   // GBK_TO_UNICODE[4429] := 16#5C32;
   // GBK_TO_UNICODE[4430] := 16#8CBD;
   // GBK_TO_UNICODE[4431] := 16#5C33;
   // GBK_TO_UNICODE[4432] := 16#8CBE;
   // GBK_TO_UNICODE[4433] := 16#5C35;
   // GBK_TO_UNICODE[4434] := 16#8CBF;
   // GBK_TO_UNICODE[4435] := 16#5C36;
   // GBK_TO_UNICODE[4436] := 16#8CC0;
   // GBK_TO_UNICODE[4437] := 16#5C37;
   // GBK_TO_UNICODE[4438] := 16#8CC1;
   // GBK_TO_UNICODE[4439] := 16#5C43;
   // GBK_TO_UNICODE[4440] := 16#8CC2;
   // GBK_TO_UNICODE[4441] := 16#5C44;
   // GBK_TO_UNICODE[4442] := 16#8CC3;
   // GBK_TO_UNICODE[4443] := 16#5C46;
   // GBK_TO_UNICODE[4444] := 16#8CC4;
   // GBK_TO_UNICODE[4445] := 16#5C47;
   // GBK_TO_UNICODE[4446] := 16#8CC5;
   // GBK_TO_UNICODE[4447] := 16#5C4C;
   // GBK_TO_UNICODE[4448] := 16#8CC6;
   // GBK_TO_UNICODE[4449] := 16#5C4D;
   // GBK_TO_UNICODE[4450] := 16#8CC7;
   // GBK_TO_UNICODE[4451] := 16#5C52;
   // GBK_TO_UNICODE[4452] := 16#8CC8;
   // GBK_TO_UNICODE[4453] := 16#5C53;
   // GBK_TO_UNICODE[4454] := 16#8CC9;
   // GBK_TO_UNICODE[4455] := 16#5C54;
   // GBK_TO_UNICODE[4456] := 16#8CCA;
   // GBK_TO_UNICODE[4457] := 16#5C56;
   // GBK_TO_UNICODE[4458] := 16#8CCB;
   // GBK_TO_UNICODE[4459] := 16#5C57;
   // GBK_TO_UNICODE[4460] := 16#8CCC;
   // GBK_TO_UNICODE[4461] := 16#5C58;
   // GBK_TO_UNICODE[4462] := 16#8CCD;
   // GBK_TO_UNICODE[4463] := 16#5C5A;
   // GBK_TO_UNICODE[4464] := 16#8CCE;
   // GBK_TO_UNICODE[4465] := 16#5C5B;
   // GBK_TO_UNICODE[4466] := 16#8CCF;
   // GBK_TO_UNICODE[4467] := 16#5C5C;
   // GBK_TO_UNICODE[4468] := 16#8CD0;
   // GBK_TO_UNICODE[4469] := 16#5C5D;
   // GBK_TO_UNICODE[4470] := 16#8CD1;
   // GBK_TO_UNICODE[4471] := 16#5C5F;
   // GBK_TO_UNICODE[4472] := 16#8CD2;
   // GBK_TO_UNICODE[4473] := 16#5C62;
   // GBK_TO_UNICODE[4474] := 16#8CD3;
   // GBK_TO_UNICODE[4475] := 16#5C64;
   // GBK_TO_UNICODE[4476] := 16#8CD4;
   // GBK_TO_UNICODE[4477] := 16#5C67;
   // GBK_TO_UNICODE[4478] := 16#8CD5;
   // GBK_TO_UNICODE[4479] := 16#5C68;
   // GBK_TO_UNICODE[4480] := 16#8CD6;
   // GBK_TO_UNICODE[4481] := 16#5C69;
   // GBK_TO_UNICODE[4482] := 16#8CD7;
   // GBK_TO_UNICODE[4483] := 16#5C6A;
   // GBK_TO_UNICODE[4484] := 16#8CD8;
   // GBK_TO_UNICODE[4485] := 16#5C6B;
   // GBK_TO_UNICODE[4486] := 16#8CD9;
   // GBK_TO_UNICODE[4487] := 16#5C6C;
   // GBK_TO_UNICODE[4488] := 16#8CDA;
   // GBK_TO_UNICODE[4489] := 16#5C6D;
   // GBK_TO_UNICODE[4490] := 16#8CDB;
   // GBK_TO_UNICODE[4491] := 16#5C70;
   // GBK_TO_UNICODE[4492] := 16#8CDC;
   // GBK_TO_UNICODE[4493] := 16#5C72;
   // GBK_TO_UNICODE[4494] := 16#8CDD;
   // GBK_TO_UNICODE[4495] := 16#5C73;
   // GBK_TO_UNICODE[4496] := 16#8CDE;
   // GBK_TO_UNICODE[4497] := 16#5C74;
   // GBK_TO_UNICODE[4498] := 16#8CDF;
   // GBK_TO_UNICODE[4499] := 16#5C75;
   // GBK_TO_UNICODE[4500] := 16#8CE0;
   // GBK_TO_UNICODE[4501] := 16#5C76;
   // GBK_TO_UNICODE[4502] := 16#8CE1;
   // GBK_TO_UNICODE[4503] := 16#5C77;
   // GBK_TO_UNICODE[4504] := 16#8CE2;
   // GBK_TO_UNICODE[4505] := 16#5C78;
   // GBK_TO_UNICODE[4506] := 16#8CE3;
   // GBK_TO_UNICODE[4507] := 16#5C7B;
   // GBK_TO_UNICODE[4508] := 16#8CE4;
   // GBK_TO_UNICODE[4509] := 16#5C7C;
   // GBK_TO_UNICODE[4510] := 16#8CE5;
   // GBK_TO_UNICODE[4511] := 16#5C7D;
   // GBK_TO_UNICODE[4512] := 16#8CE6;
   // GBK_TO_UNICODE[4513] := 16#5C7E;
   // GBK_TO_UNICODE[4514] := 16#8CE7;
   // GBK_TO_UNICODE[4515] := 16#5C80;
   // GBK_TO_UNICODE[4516] := 16#8CE8;
   // GBK_TO_UNICODE[4517] := 16#5C83;
   // GBK_TO_UNICODE[4518] := 16#8CE9;
   // GBK_TO_UNICODE[4519] := 16#5C84;
   // GBK_TO_UNICODE[4520] := 16#8CEA;
   // GBK_TO_UNICODE[4521] := 16#5C85;
   // GBK_TO_UNICODE[4522] := 16#8CEB;
   // GBK_TO_UNICODE[4523] := 16#5C86;
   // GBK_TO_UNICODE[4524] := 16#8CEC;
   // GBK_TO_UNICODE[4525] := 16#5C87;
   // GBK_TO_UNICODE[4526] := 16#8CED;
   // GBK_TO_UNICODE[4527] := 16#5C89;
   // GBK_TO_UNICODE[4528] := 16#8CEE;
   // GBK_TO_UNICODE[4529] := 16#5C8A;
   // GBK_TO_UNICODE[4530] := 16#8CEF;
   // GBK_TO_UNICODE[4531] := 16#5C8B;
   // GBK_TO_UNICODE[4532] := 16#8CF0;
   // GBK_TO_UNICODE[4533] := 16#5C8E;
   // GBK_TO_UNICODE[4534] := 16#8CF1;
   // GBK_TO_UNICODE[4535] := 16#5C8F;
   // GBK_TO_UNICODE[4536] := 16#8CF2;
   // GBK_TO_UNICODE[4537] := 16#5C92;
   // GBK_TO_UNICODE[4538] := 16#8CF3;
   // GBK_TO_UNICODE[4539] := 16#5C93;
   // GBK_TO_UNICODE[4540] := 16#8CF4;
   // GBK_TO_UNICODE[4541] := 16#5C95;
   // GBK_TO_UNICODE[4542] := 16#8CF5;
   // GBK_TO_UNICODE[4543] := 16#5C9D;
   // GBK_TO_UNICODE[4544] := 16#8CF6;
   // GBK_TO_UNICODE[4545] := 16#5C9E;
   // GBK_TO_UNICODE[4546] := 16#8CF7;
   // GBK_TO_UNICODE[4547] := 16#5C9F;
   // GBK_TO_UNICODE[4548] := 16#8CF8;
   // GBK_TO_UNICODE[4549] := 16#5CA0;
   // GBK_TO_UNICODE[4550] := 16#8CF9;
   // GBK_TO_UNICODE[4551] := 16#5CA1;
   // GBK_TO_UNICODE[4552] := 16#8CFA;
   // GBK_TO_UNICODE[4553] := 16#5CA4;
   // GBK_TO_UNICODE[4554] := 16#8CFB;
   // GBK_TO_UNICODE[4555] := 16#5CA5;
   // GBK_TO_UNICODE[4556] := 16#8CFC;
   // GBK_TO_UNICODE[4557] := 16#5CA6;
   // GBK_TO_UNICODE[4558] := 16#8CFD;
   // GBK_TO_UNICODE[4559] := 16#5CA7;
   // GBK_TO_UNICODE[4560] := 16#8CFE;
   // GBK_TO_UNICODE[4561] := 16#5CA8;
   // GBK_TO_UNICODE[4562] := 16#8D40;
   // GBK_TO_UNICODE[4563] := 16#5CAA;
   // GBK_TO_UNICODE[4564] := 16#8D41;
   // GBK_TO_UNICODE[4565] := 16#5CAE;
   // GBK_TO_UNICODE[4566] := 16#8D42;
   // GBK_TO_UNICODE[4567] := 16#5CAF;
   // GBK_TO_UNICODE[4568] := 16#8D43;
   // GBK_TO_UNICODE[4569] := 16#5CB0;
   // GBK_TO_UNICODE[4570] := 16#8D44;
   // GBK_TO_UNICODE[4571] := 16#5CB2;
   // GBK_TO_UNICODE[4572] := 16#8D45;
   // GBK_TO_UNICODE[4573] := 16#5CB4;
   // GBK_TO_UNICODE[4574] := 16#8D46;
   // GBK_TO_UNICODE[4575] := 16#5CB6;
   // GBK_TO_UNICODE[4576] := 16#8D47;
   // GBK_TO_UNICODE[4577] := 16#5CB9;
   // GBK_TO_UNICODE[4578] := 16#8D48;
   // GBK_TO_UNICODE[4579] := 16#5CBA;
   // GBK_TO_UNICODE[4580] := 16#8D49;
   // GBK_TO_UNICODE[4581] := 16#5CBB;
   // GBK_TO_UNICODE[4582] := 16#8D4A;
   // GBK_TO_UNICODE[4583] := 16#5CBC;
   // GBK_TO_UNICODE[4584] := 16#8D4B;
   // GBK_TO_UNICODE[4585] := 16#5CBE;
   // GBK_TO_UNICODE[4586] := 16#8D4C;
   // GBK_TO_UNICODE[4587] := 16#5CC0;
   // GBK_TO_UNICODE[4588] := 16#8D4D;
   // GBK_TO_UNICODE[4589] := 16#5CC2;
   // GBK_TO_UNICODE[4590] := 16#8D4E;
   // GBK_TO_UNICODE[4591] := 16#5CC3;
   // GBK_TO_UNICODE[4592] := 16#8D4F;
   // GBK_TO_UNICODE[4593] := 16#5CC5;
   // GBK_TO_UNICODE[4594] := 16#8D50;
   // GBK_TO_UNICODE[4595] := 16#5CC6;
   // GBK_TO_UNICODE[4596] := 16#8D51;
   // GBK_TO_UNICODE[4597] := 16#5CC7;
   // GBK_TO_UNICODE[4598] := 16#8D52;
   // GBK_TO_UNICODE[4599] := 16#5CC8;
   // GBK_TO_UNICODE[4600] := 16#8D53;
   // GBK_TO_UNICODE[4601] := 16#5CC9;
   // GBK_TO_UNICODE[4602] := 16#8D54;
   // GBK_TO_UNICODE[4603] := 16#5CCA;
   // GBK_TO_UNICODE[4604] := 16#8D55;
   // GBK_TO_UNICODE[4605] := 16#5CCC;
   // GBK_TO_UNICODE[4606] := 16#8D56;
   // GBK_TO_UNICODE[4607] := 16#5CCD;
   // GBK_TO_UNICODE[4608] := 16#8D57;
   // GBK_TO_UNICODE[4609] := 16#5CCE;
   // GBK_TO_UNICODE[4610] := 16#8D58;
   // GBK_TO_UNICODE[4611] := 16#5CCF;
   // GBK_TO_UNICODE[4612] := 16#8D59;
   // GBK_TO_UNICODE[4613] := 16#5CD0;
   // GBK_TO_UNICODE[4614] := 16#8D5A;
   // GBK_TO_UNICODE[4615] := 16#5CD1;
   // GBK_TO_UNICODE[4616] := 16#8D5B;
   // GBK_TO_UNICODE[4617] := 16#5CD3;
   // GBK_TO_UNICODE[4618] := 16#8D5C;
   // GBK_TO_UNICODE[4619] := 16#5CD4;
   // GBK_TO_UNICODE[4620] := 16#8D5D;
   // GBK_TO_UNICODE[4621] := 16#5CD5;
   // GBK_TO_UNICODE[4622] := 16#8D5E;
   // GBK_TO_UNICODE[4623] := 16#5CD6;
   // GBK_TO_UNICODE[4624] := 16#8D5F;
   // GBK_TO_UNICODE[4625] := 16#5CD7;
   // GBK_TO_UNICODE[4626] := 16#8D60;
   // GBK_TO_UNICODE[4627] := 16#5CD8;
   // GBK_TO_UNICODE[4628] := 16#8D61;
   // GBK_TO_UNICODE[4629] := 16#5CDA;
   // GBK_TO_UNICODE[4630] := 16#8D62;
   // GBK_TO_UNICODE[4631] := 16#5CDB;
   // GBK_TO_UNICODE[4632] := 16#8D63;
   // GBK_TO_UNICODE[4633] := 16#5CDC;
   // GBK_TO_UNICODE[4634] := 16#8D64;
   // GBK_TO_UNICODE[4635] := 16#5CDD;
   // GBK_TO_UNICODE[4636] := 16#8D65;
   // GBK_TO_UNICODE[4637] := 16#5CDE;
   // GBK_TO_UNICODE[4638] := 16#8D66;
   // GBK_TO_UNICODE[4639] := 16#5CDF;
   // GBK_TO_UNICODE[4640] := 16#8D67;
   // GBK_TO_UNICODE[4641] := 16#5CE0;
   // GBK_TO_UNICODE[4642] := 16#8D68;
   // GBK_TO_UNICODE[4643] := 16#5CE2;
   // GBK_TO_UNICODE[4644] := 16#8D69;
   // GBK_TO_UNICODE[4645] := 16#5CE3;
   // GBK_TO_UNICODE[4646] := 16#8D6A;
   // GBK_TO_UNICODE[4647] := 16#5CE7;
   // GBK_TO_UNICODE[4648] := 16#8D6B;
   // GBK_TO_UNICODE[4649] := 16#5CE9;
   // GBK_TO_UNICODE[4650] := 16#8D6C;
   // GBK_TO_UNICODE[4651] := 16#5CEB;
   // GBK_TO_UNICODE[4652] := 16#8D6D;
   // GBK_TO_UNICODE[4653] := 16#5CEC;
   // GBK_TO_UNICODE[4654] := 16#8D6E;
   // GBK_TO_UNICODE[4655] := 16#5CEE;
   // GBK_TO_UNICODE[4656] := 16#8D6F;
   // GBK_TO_UNICODE[4657] := 16#5CEF;
   // GBK_TO_UNICODE[4658] := 16#8D70;
   // GBK_TO_UNICODE[4659] := 16#5CF1;
   // GBK_TO_UNICODE[4660] := 16#8D71;
   // GBK_TO_UNICODE[4661] := 16#5CF2;
   // GBK_TO_UNICODE[4662] := 16#8D72;
   // GBK_TO_UNICODE[4663] := 16#5CF3;
   // GBK_TO_UNICODE[4664] := 16#8D73;
   // GBK_TO_UNICODE[4665] := 16#5CF4;
   // GBK_TO_UNICODE[4666] := 16#8D74;
   // GBK_TO_UNICODE[4667] := 16#5CF5;
   // GBK_TO_UNICODE[4668] := 16#8D75;
   // GBK_TO_UNICODE[4669] := 16#5CF6;
   // GBK_TO_UNICODE[4670] := 16#8D76;
   // GBK_TO_UNICODE[4671] := 16#5CF7;
   // GBK_TO_UNICODE[4672] := 16#8D77;
   // GBK_TO_UNICODE[4673] := 16#5CF8;
   // GBK_TO_UNICODE[4674] := 16#8D78;
   // GBK_TO_UNICODE[4675] := 16#5CF9;
   // GBK_TO_UNICODE[4676] := 16#8D79;
   // GBK_TO_UNICODE[4677] := 16#5CFA;
   // GBK_TO_UNICODE[4678] := 16#8D7A;
   // GBK_TO_UNICODE[4679] := 16#5CFC;
   // GBK_TO_UNICODE[4680] := 16#8D7B;
   // GBK_TO_UNICODE[4681] := 16#5CFD;
   // GBK_TO_UNICODE[4682] := 16#8D7C;
   // GBK_TO_UNICODE[4683] := 16#5CFE;
   // GBK_TO_UNICODE[4684] := 16#8D7D;
   // GBK_TO_UNICODE[4685] := 16#5CFF;
   // GBK_TO_UNICODE[4686] := 16#8D7E;
   // GBK_TO_UNICODE[4687] := 16#5D00;
   // GBK_TO_UNICODE[4688] := 16#8D80;
   // GBK_TO_UNICODE[4689] := 16#5D01;
   // GBK_TO_UNICODE[4690] := 16#8D81;
   // GBK_TO_UNICODE[4691] := 16#5D04;
   // GBK_TO_UNICODE[4692] := 16#8D82;
   // GBK_TO_UNICODE[4693] := 16#5D05;
   // GBK_TO_UNICODE[4694] := 16#8D83;
   // GBK_TO_UNICODE[4695] := 16#5D08;
   // GBK_TO_UNICODE[4696] := 16#8D84;
   // GBK_TO_UNICODE[4697] := 16#5D09;
   // GBK_TO_UNICODE[4698] := 16#8D85;
   // GBK_TO_UNICODE[4699] := 16#5D0A;
   // GBK_TO_UNICODE[4700] := 16#8D86;
   // GBK_TO_UNICODE[4701] := 16#5D0B;
   // GBK_TO_UNICODE[4702] := 16#8D87;
   // GBK_TO_UNICODE[4703] := 16#5D0C;
   // GBK_TO_UNICODE[4704] := 16#8D88;
   // GBK_TO_UNICODE[4705] := 16#5D0D;
   // GBK_TO_UNICODE[4706] := 16#8D89;
   // GBK_TO_UNICODE[4707] := 16#5D0F;
   // GBK_TO_UNICODE[4708] := 16#8D8A;
   // GBK_TO_UNICODE[4709] := 16#5D10;
   // GBK_TO_UNICODE[4710] := 16#8D8B;
   // GBK_TO_UNICODE[4711] := 16#5D11;
   // GBK_TO_UNICODE[4712] := 16#8D8C;
   // GBK_TO_UNICODE[4713] := 16#5D12;
   // GBK_TO_UNICODE[4714] := 16#8D8D;
   // GBK_TO_UNICODE[4715] := 16#5D13;
   // GBK_TO_UNICODE[4716] := 16#8D8E;
   // GBK_TO_UNICODE[4717] := 16#5D15;
   // GBK_TO_UNICODE[4718] := 16#8D8F;
   // GBK_TO_UNICODE[4719] := 16#5D17;
   // GBK_TO_UNICODE[4720] := 16#8D90;
   // GBK_TO_UNICODE[4721] := 16#5D18;
   // GBK_TO_UNICODE[4722] := 16#8D91;
   // GBK_TO_UNICODE[4723] := 16#5D19;
   // GBK_TO_UNICODE[4724] := 16#8D92;
   // GBK_TO_UNICODE[4725] := 16#5D1A;
   // GBK_TO_UNICODE[4726] := 16#8D93;
   // GBK_TO_UNICODE[4727] := 16#5D1C;
   // GBK_TO_UNICODE[4728] := 16#8D94;
   // GBK_TO_UNICODE[4729] := 16#5D1D;
   // GBK_TO_UNICODE[4730] := 16#8D95;
   // GBK_TO_UNICODE[4731] := 16#5D1F;
   // GBK_TO_UNICODE[4732] := 16#8D96;
   // GBK_TO_UNICODE[4733] := 16#5D20;
   // GBK_TO_UNICODE[4734] := 16#8D97;
   // GBK_TO_UNICODE[4735] := 16#5D21;
   // GBK_TO_UNICODE[4736] := 16#8D98;
   // GBK_TO_UNICODE[4737] := 16#5D22;
   // GBK_TO_UNICODE[4738] := 16#8D99;
   // GBK_TO_UNICODE[4739] := 16#5D23;
   // GBK_TO_UNICODE[4740] := 16#8D9A;
   // GBK_TO_UNICODE[4741] := 16#5D25;
   // GBK_TO_UNICODE[4742] := 16#8D9B;
   // GBK_TO_UNICODE[4743] := 16#5D28;
   // GBK_TO_UNICODE[4744] := 16#8D9C;
   // GBK_TO_UNICODE[4745] := 16#5D2A;
   // GBK_TO_UNICODE[4746] := 16#8D9D;
   // GBK_TO_UNICODE[4747] := 16#5D2B;
   // GBK_TO_UNICODE[4748] := 16#8D9E;
   // GBK_TO_UNICODE[4749] := 16#5D2C;
   // GBK_TO_UNICODE[4750] := 16#8D9F;
   // GBK_TO_UNICODE[4751] := 16#5D2F;
   // GBK_TO_UNICODE[4752] := 16#8DA0;
   // GBK_TO_UNICODE[4753] := 16#5D30;
   // GBK_TO_UNICODE[4754] := 16#8DA1;
   // GBK_TO_UNICODE[4755] := 16#5D31;
   // GBK_TO_UNICODE[4756] := 16#8DA2;
   // GBK_TO_UNICODE[4757] := 16#5D32;
   // GBK_TO_UNICODE[4758] := 16#8DA3;
   // GBK_TO_UNICODE[4759] := 16#5D33;
   // GBK_TO_UNICODE[4760] := 16#8DA4;
   // GBK_TO_UNICODE[4761] := 16#5D35;
   // GBK_TO_UNICODE[4762] := 16#8DA5;
   // GBK_TO_UNICODE[4763] := 16#5D36;
   // GBK_TO_UNICODE[4764] := 16#8DA6;
   // GBK_TO_UNICODE[4765] := 16#5D37;
   // GBK_TO_UNICODE[4766] := 16#8DA7;
   // GBK_TO_UNICODE[4767] := 16#5D38;
   // GBK_TO_UNICODE[4768] := 16#8DA8;
   // GBK_TO_UNICODE[4769] := 16#5D39;
   // GBK_TO_UNICODE[4770] := 16#8DA9;
   // GBK_TO_UNICODE[4771] := 16#5D3A;
   // GBK_TO_UNICODE[4772] := 16#8DAA;
   // GBK_TO_UNICODE[4773] := 16#5D3B;
   // GBK_TO_UNICODE[4774] := 16#8DAB;
   // GBK_TO_UNICODE[4775] := 16#5D3C;
   // GBK_TO_UNICODE[4776] := 16#8DAC;
   // GBK_TO_UNICODE[4777] := 16#5D3F;
   // GBK_TO_UNICODE[4778] := 16#8DAD;
   // GBK_TO_UNICODE[4779] := 16#5D40;
   // GBK_TO_UNICODE[4780] := 16#8DAE;
   // GBK_TO_UNICODE[4781] := 16#5D41;
   // GBK_TO_UNICODE[4782] := 16#8DAF;
   // GBK_TO_UNICODE[4783] := 16#5D42;
   // GBK_TO_UNICODE[4784] := 16#8DB0;
   // GBK_TO_UNICODE[4785] := 16#5D43;
   // GBK_TO_UNICODE[4786] := 16#8DB1;
   // GBK_TO_UNICODE[4787] := 16#5D44;
   // GBK_TO_UNICODE[4788] := 16#8DB2;
   // GBK_TO_UNICODE[4789] := 16#5D45;
   // GBK_TO_UNICODE[4790] := 16#8DB3;
   // GBK_TO_UNICODE[4791] := 16#5D46;
   // GBK_TO_UNICODE[4792] := 16#8DB4;
   // GBK_TO_UNICODE[4793] := 16#5D48;
   // GBK_TO_UNICODE[4794] := 16#8DB5;
   // GBK_TO_UNICODE[4795] := 16#5D49;
   // GBK_TO_UNICODE[4796] := 16#8DB6;
   // GBK_TO_UNICODE[4797] := 16#5D4D;
   // GBK_TO_UNICODE[4798] := 16#8DB7;
   // GBK_TO_UNICODE[4799] := 16#5D4E;
   // GBK_TO_UNICODE[4800] := 16#8DB8;
   // GBK_TO_UNICODE[4801] := 16#5D4F;
   // GBK_TO_UNICODE[4802] := 16#8DB9;
   // GBK_TO_UNICODE[4803] := 16#5D50;
   // GBK_TO_UNICODE[4804] := 16#8DBA;
   // GBK_TO_UNICODE[4805] := 16#5D51;
   // GBK_TO_UNICODE[4806] := 16#8DBB;
   // GBK_TO_UNICODE[4807] := 16#5D52;
   // GBK_TO_UNICODE[4808] := 16#8DBC;
   // GBK_TO_UNICODE[4809] := 16#5D53;
   // GBK_TO_UNICODE[4810] := 16#8DBD;
   // GBK_TO_UNICODE[4811] := 16#5D54;
   // GBK_TO_UNICODE[4812] := 16#8DBE;
   // GBK_TO_UNICODE[4813] := 16#5D55;
   // GBK_TO_UNICODE[4814] := 16#8DBF;
   // GBK_TO_UNICODE[4815] := 16#5D56;
   // GBK_TO_UNICODE[4816] := 16#8DC0;
   // GBK_TO_UNICODE[4817] := 16#5D57;
   // GBK_TO_UNICODE[4818] := 16#8DC1;
   // GBK_TO_UNICODE[4819] := 16#5D59;
   // GBK_TO_UNICODE[4820] := 16#8DC2;
   // GBK_TO_UNICODE[4821] := 16#5D5A;
   // GBK_TO_UNICODE[4822] := 16#8DC3;
   // GBK_TO_UNICODE[4823] := 16#5D5C;
   // GBK_TO_UNICODE[4824] := 16#8DC4;
   // GBK_TO_UNICODE[4825] := 16#5D5E;
   // GBK_TO_UNICODE[4826] := 16#8DC5;
   // GBK_TO_UNICODE[4827] := 16#5D5F;
   // GBK_TO_UNICODE[4828] := 16#8DC6;
   // GBK_TO_UNICODE[4829] := 16#5D60;
   // GBK_TO_UNICODE[4830] := 16#8DC7;
   // GBK_TO_UNICODE[4831] := 16#5D61;
   // GBK_TO_UNICODE[4832] := 16#8DC8;
   // GBK_TO_UNICODE[4833] := 16#5D62;
   // GBK_TO_UNICODE[4834] := 16#8DC9;
   // GBK_TO_UNICODE[4835] := 16#5D63;
   // GBK_TO_UNICODE[4836] := 16#8DCA;
   // GBK_TO_UNICODE[4837] := 16#5D64;
   // GBK_TO_UNICODE[4838] := 16#8DCB;
   // GBK_TO_UNICODE[4839] := 16#5D65;
   // GBK_TO_UNICODE[4840] := 16#8DCC;
   // GBK_TO_UNICODE[4841] := 16#5D66;
   // GBK_TO_UNICODE[4842] := 16#8DCD;
   // GBK_TO_UNICODE[4843] := 16#5D67;
   // GBK_TO_UNICODE[4844] := 16#8DCE;
   // GBK_TO_UNICODE[4845] := 16#5D68;
   // GBK_TO_UNICODE[4846] := 16#8DCF;
   // GBK_TO_UNICODE[4847] := 16#5D6A;
   // GBK_TO_UNICODE[4848] := 16#8DD0;
   // GBK_TO_UNICODE[4849] := 16#5D6D;
   // GBK_TO_UNICODE[4850] := 16#8DD1;
   // GBK_TO_UNICODE[4851] := 16#5D6E;
   // GBK_TO_UNICODE[4852] := 16#8DD2;
   // GBK_TO_UNICODE[4853] := 16#5D70;
   // GBK_TO_UNICODE[4854] := 16#8DD3;
   // GBK_TO_UNICODE[4855] := 16#5D71;
   // GBK_TO_UNICODE[4856] := 16#8DD4;
   // GBK_TO_UNICODE[4857] := 16#5D72;
   // GBK_TO_UNICODE[4858] := 16#8DD5;
   // GBK_TO_UNICODE[4859] := 16#5D73;
   // GBK_TO_UNICODE[4860] := 16#8DD6;
   // GBK_TO_UNICODE[4861] := 16#5D75;
   // GBK_TO_UNICODE[4862] := 16#8DD7;
   // GBK_TO_UNICODE[4863] := 16#5D76;
   // GBK_TO_UNICODE[4864] := 16#8DD8;
   // GBK_TO_UNICODE[4865] := 16#5D77;
   // GBK_TO_UNICODE[4866] := 16#8DD9;
   // GBK_TO_UNICODE[4867] := 16#5D78;
   // GBK_TO_UNICODE[4868] := 16#8DDA;
   // GBK_TO_UNICODE[4869] := 16#5D79;
   // GBK_TO_UNICODE[4870] := 16#8DDB;
   // GBK_TO_UNICODE[4871] := 16#5D7A;
   // GBK_TO_UNICODE[4872] := 16#8DDC;
   // GBK_TO_UNICODE[4873] := 16#5D7B;
   // GBK_TO_UNICODE[4874] := 16#8DDD;
   // GBK_TO_UNICODE[4875] := 16#5D7C;
   // GBK_TO_UNICODE[4876] := 16#8DDE;
   // GBK_TO_UNICODE[4877] := 16#5D7D;
   // GBK_TO_UNICODE[4878] := 16#8DDF;
   // GBK_TO_UNICODE[4879] := 16#5D7E;
   // GBK_TO_UNICODE[4880] := 16#8DE0;
   // GBK_TO_UNICODE[4881] := 16#5D7F;
   // GBK_TO_UNICODE[4882] := 16#8DE1;
   // GBK_TO_UNICODE[4883] := 16#5D80;
   // GBK_TO_UNICODE[4884] := 16#8DE2;
   // GBK_TO_UNICODE[4885] := 16#5D81;
   // GBK_TO_UNICODE[4886] := 16#8DE3;
   // GBK_TO_UNICODE[4887] := 16#5D83;
   // GBK_TO_UNICODE[4888] := 16#8DE4;
   // GBK_TO_UNICODE[4889] := 16#5D84;
   // GBK_TO_UNICODE[4890] := 16#8DE5;
   // GBK_TO_UNICODE[4891] := 16#5D85;
   // GBK_TO_UNICODE[4892] := 16#8DE6;
   // GBK_TO_UNICODE[4893] := 16#5D86;
   // GBK_TO_UNICODE[4894] := 16#8DE7;
   // GBK_TO_UNICODE[4895] := 16#5D87;
   // GBK_TO_UNICODE[4896] := 16#8DE8;
   // GBK_TO_UNICODE[4897] := 16#5D88;
   // GBK_TO_UNICODE[4898] := 16#8DE9;
   // GBK_TO_UNICODE[4899] := 16#5D89;
   // GBK_TO_UNICODE[4900] := 16#8DEA;
   // GBK_TO_UNICODE[4901] := 16#5D8A;
   // GBK_TO_UNICODE[4902] := 16#8DEB;
   // GBK_TO_UNICODE[4903] := 16#5D8B;
   // GBK_TO_UNICODE[4904] := 16#8DEC;
   // GBK_TO_UNICODE[4905] := 16#5D8C;
   // GBK_TO_UNICODE[4906] := 16#8DED;
   // GBK_TO_UNICODE[4907] := 16#5D8D;
   // GBK_TO_UNICODE[4908] := 16#8DEE;
   // GBK_TO_UNICODE[4909] := 16#5D8E;
   // GBK_TO_UNICODE[4910] := 16#8DEF;
   // GBK_TO_UNICODE[4911] := 16#5D8F;
   // GBK_TO_UNICODE[4912] := 16#8DF0;
   // GBK_TO_UNICODE[4913] := 16#5D90;
   // GBK_TO_UNICODE[4914] := 16#8DF1;
   // GBK_TO_UNICODE[4915] := 16#5D91;
   // GBK_TO_UNICODE[4916] := 16#8DF2;
   // GBK_TO_UNICODE[4917] := 16#5D92;
   // GBK_TO_UNICODE[4918] := 16#8DF3;
   // GBK_TO_UNICODE[4919] := 16#5D93;
   // GBK_TO_UNICODE[4920] := 16#8DF4;
   // GBK_TO_UNICODE[4921] := 16#5D94;
   // GBK_TO_UNICODE[4922] := 16#8DF5;
   // GBK_TO_UNICODE[4923] := 16#5D95;
   // GBK_TO_UNICODE[4924] := 16#8DF6;
   // GBK_TO_UNICODE[4925] := 16#5D96;
   // GBK_TO_UNICODE[4926] := 16#8DF7;
   // GBK_TO_UNICODE[4927] := 16#5D97;
   // GBK_TO_UNICODE[4928] := 16#8DF8;
   // GBK_TO_UNICODE[4929] := 16#5D98;
   // GBK_TO_UNICODE[4930] := 16#8DF9;
   // GBK_TO_UNICODE[4931] := 16#5D9A;
   // GBK_TO_UNICODE[4932] := 16#8DFA;
   // GBK_TO_UNICODE[4933] := 16#5D9B;
   // GBK_TO_UNICODE[4934] := 16#8DFB;
   // GBK_TO_UNICODE[4935] := 16#5D9C;
   // GBK_TO_UNICODE[4936] := 16#8DFC;
   // GBK_TO_UNICODE[4937] := 16#5D9E;
   // GBK_TO_UNICODE[4938] := 16#8DFD;
   // GBK_TO_UNICODE[4939] := 16#5D9F;
   // GBK_TO_UNICODE[4940] := 16#8DFE;
   // GBK_TO_UNICODE[4941] := 16#5DA0;
   // GBK_TO_UNICODE[4942] := 16#8E40;
   // GBK_TO_UNICODE[4943] := 16#5DA1;
   // GBK_TO_UNICODE[4944] := 16#8E41;
   // GBK_TO_UNICODE[4945] := 16#5DA2;
   // GBK_TO_UNICODE[4946] := 16#8E42;
   // GBK_TO_UNICODE[4947] := 16#5DA3;
   // GBK_TO_UNICODE[4948] := 16#8E43;
   // GBK_TO_UNICODE[4949] := 16#5DA4;
   // GBK_TO_UNICODE[4950] := 16#8E44;
   // GBK_TO_UNICODE[4951] := 16#5DA5;
   // GBK_TO_UNICODE[4952] := 16#8E45;
   // GBK_TO_UNICODE[4953] := 16#5DA6;
   // GBK_TO_UNICODE[4954] := 16#8E46;
   // GBK_TO_UNICODE[4955] := 16#5DA7;
   // GBK_TO_UNICODE[4956] := 16#8E47;
   // GBK_TO_UNICODE[4957] := 16#5DA8;
   // GBK_TO_UNICODE[4958] := 16#8E48;
   // GBK_TO_UNICODE[4959] := 16#5DA9;
   // GBK_TO_UNICODE[4960] := 16#8E49;
   // GBK_TO_UNICODE[4961] := 16#5DAA;
   // GBK_TO_UNICODE[4962] := 16#8E4A;
   // GBK_TO_UNICODE[4963] := 16#5DAB;
   // GBK_TO_UNICODE[4964] := 16#8E4B;
   // GBK_TO_UNICODE[4965] := 16#5DAC;
   // GBK_TO_UNICODE[4966] := 16#8E4C;
   // GBK_TO_UNICODE[4967] := 16#5DAD;
   // GBK_TO_UNICODE[4968] := 16#8E4D;
   // GBK_TO_UNICODE[4969] := 16#5DAE;
   // GBK_TO_UNICODE[4970] := 16#8E4E;
   // GBK_TO_UNICODE[4971] := 16#5DAF;
   // GBK_TO_UNICODE[4972] := 16#8E4F;
   // GBK_TO_UNICODE[4973] := 16#5DB0;
   // GBK_TO_UNICODE[4974] := 16#8E50;
   // GBK_TO_UNICODE[4975] := 16#5DB1;
   // GBK_TO_UNICODE[4976] := 16#8E51;
   // GBK_TO_UNICODE[4977] := 16#5DB2;
   // GBK_TO_UNICODE[4978] := 16#8E52;
   // GBK_TO_UNICODE[4979] := 16#5DB3;
   // GBK_TO_UNICODE[4980] := 16#8E53;
   // GBK_TO_UNICODE[4981] := 16#5DB4;
   // GBK_TO_UNICODE[4982] := 16#8E54;
   // GBK_TO_UNICODE[4983] := 16#5DB5;
   // GBK_TO_UNICODE[4984] := 16#8E55;
   // GBK_TO_UNICODE[4985] := 16#5DB6;
   // GBK_TO_UNICODE[4986] := 16#8E56;
   // GBK_TO_UNICODE[4987] := 16#5DB8;
   // GBK_TO_UNICODE[4988] := 16#8E57;
   // GBK_TO_UNICODE[4989] := 16#5DB9;
   // GBK_TO_UNICODE[4990] := 16#8E58;
   // GBK_TO_UNICODE[4991] := 16#5DBA;
   // GBK_TO_UNICODE[4992] := 16#8E59;
   // GBK_TO_UNICODE[4993] := 16#5DBB;
   // GBK_TO_UNICODE[4994] := 16#8E5A;
   // GBK_TO_UNICODE[4995] := 16#5DBC;
   // GBK_TO_UNICODE[4996] := 16#8E5B;
   // GBK_TO_UNICODE[4997] := 16#5DBD;
   // GBK_TO_UNICODE[4998] := 16#8E5C;
   // GBK_TO_UNICODE[4999] := 16#5DBE;
   // GBK_TO_UNICODE[5000] := 16#8E5D;
   // GBK_TO_UNICODE[5001] := 16#5DBF;
   // GBK_TO_UNICODE[5002] := 16#8E5E;
   // GBK_TO_UNICODE[5003] := 16#5DC0;
   // GBK_TO_UNICODE[5004] := 16#8E5F;
   // GBK_TO_UNICODE[5005] := 16#5DC1;
   // GBK_TO_UNICODE[5006] := 16#8E60;
   // GBK_TO_UNICODE[5007] := 16#5DC2;
   // GBK_TO_UNICODE[5008] := 16#8E61;
   // GBK_TO_UNICODE[5009] := 16#5DC3;
   // GBK_TO_UNICODE[5010] := 16#8E62;
   // GBK_TO_UNICODE[5011] := 16#5DC4;
   // GBK_TO_UNICODE[5012] := 16#8E63;
   // GBK_TO_UNICODE[5013] := 16#5DC6;
   // GBK_TO_UNICODE[5014] := 16#8E64;
   // GBK_TO_UNICODE[5015] := 16#5DC7;
   // GBK_TO_UNICODE[5016] := 16#8E65;
   // GBK_TO_UNICODE[5017] := 16#5DC8;
   // GBK_TO_UNICODE[5018] := 16#8E66;
   // GBK_TO_UNICODE[5019] := 16#5DC9;
   // GBK_TO_UNICODE[5020] := 16#8E67;
   // GBK_TO_UNICODE[5021] := 16#5DCA;
   // GBK_TO_UNICODE[5022] := 16#8E68;
   // GBK_TO_UNICODE[5023] := 16#5DCB;
   // GBK_TO_UNICODE[5024] := 16#8E69;
   // GBK_TO_UNICODE[5025] := 16#5DCC;
   // GBK_TO_UNICODE[5026] := 16#8E6A;
   // GBK_TO_UNICODE[5027] := 16#5DCE;
   // GBK_TO_UNICODE[5028] := 16#8E6B;
   // GBK_TO_UNICODE[5029] := 16#5DCF;
   // GBK_TO_UNICODE[5030] := 16#8E6C;
   // GBK_TO_UNICODE[5031] := 16#5DD0;
   // GBK_TO_UNICODE[5032] := 16#8E6D;
   // GBK_TO_UNICODE[5033] := 16#5DD1;
   // GBK_TO_UNICODE[5034] := 16#8E6E;
   // GBK_TO_UNICODE[5035] := 16#5DD2;
   // GBK_TO_UNICODE[5036] := 16#8E6F;
   // GBK_TO_UNICODE[5037] := 16#5DD3;
   // GBK_TO_UNICODE[5038] := 16#8E70;
   // GBK_TO_UNICODE[5039] := 16#5DD4;
   // GBK_TO_UNICODE[5040] := 16#8E71;
   // GBK_TO_UNICODE[5041] := 16#5DD5;
   // GBK_TO_UNICODE[5042] := 16#8E72;
   // GBK_TO_UNICODE[5043] := 16#5DD6;
   // GBK_TO_UNICODE[5044] := 16#8E73;
   // GBK_TO_UNICODE[5045] := 16#5DD7;
   // GBK_TO_UNICODE[5046] := 16#8E74;
   // GBK_TO_UNICODE[5047] := 16#5DD8;
   // GBK_TO_UNICODE[5048] := 16#8E75;
   // GBK_TO_UNICODE[5049] := 16#5DD9;
   // GBK_TO_UNICODE[5050] := 16#8E76;
   // GBK_TO_UNICODE[5051] := 16#5DDA;
   // GBK_TO_UNICODE[5052] := 16#8E77;
   // GBK_TO_UNICODE[5053] := 16#5DDC;
   // GBK_TO_UNICODE[5054] := 16#8E78;
   // GBK_TO_UNICODE[5055] := 16#5DDF;
   // GBK_TO_UNICODE[5056] := 16#8E79;
   // GBK_TO_UNICODE[5057] := 16#5DE0;
   // GBK_TO_UNICODE[5058] := 16#8E7A;
   // GBK_TO_UNICODE[5059] := 16#5DE3;
   // GBK_TO_UNICODE[5060] := 16#8E7B;
   // GBK_TO_UNICODE[5061] := 16#5DE4;
   // GBK_TO_UNICODE[5062] := 16#8E7C;
   // GBK_TO_UNICODE[5063] := 16#5DEA;
   // GBK_TO_UNICODE[5064] := 16#8E7D;
   // GBK_TO_UNICODE[5065] := 16#5DEC;
   // GBK_TO_UNICODE[5066] := 16#8E7E;
   // GBK_TO_UNICODE[5067] := 16#5DED;
   // GBK_TO_UNICODE[5068] := 16#8E80;
   // GBK_TO_UNICODE[5069] := 16#5DF0;
   // GBK_TO_UNICODE[5070] := 16#8E81;
   // GBK_TO_UNICODE[5071] := 16#5DF5;
   // GBK_TO_UNICODE[5072] := 16#8E82;
   // GBK_TO_UNICODE[5073] := 16#5DF6;
   // GBK_TO_UNICODE[5074] := 16#8E83;
   // GBK_TO_UNICODE[5075] := 16#5DF8;
   // GBK_TO_UNICODE[5076] := 16#8E84;
   // GBK_TO_UNICODE[5077] := 16#5DF9;
   // GBK_TO_UNICODE[5078] := 16#8E85;
   // GBK_TO_UNICODE[5079] := 16#5DFA;
   // GBK_TO_UNICODE[5080] := 16#8E86;
   // GBK_TO_UNICODE[5081] := 16#5DFB;
   // GBK_TO_UNICODE[5082] := 16#8E87;
   // GBK_TO_UNICODE[5083] := 16#5DFC;
   // GBK_TO_UNICODE[5084] := 16#8E88;
   // GBK_TO_UNICODE[5085] := 16#5DFF;
   // GBK_TO_UNICODE[5086] := 16#8E89;
   // GBK_TO_UNICODE[5087] := 16#5E00;
   // GBK_TO_UNICODE[5088] := 16#8E8A;
   // GBK_TO_UNICODE[5089] := 16#5E04;
   // GBK_TO_UNICODE[5090] := 16#8E8B;
   // GBK_TO_UNICODE[5091] := 16#5E07;
   // GBK_TO_UNICODE[5092] := 16#8E8C;
   // GBK_TO_UNICODE[5093] := 16#5E09;
   // GBK_TO_UNICODE[5094] := 16#8E8D;
   // GBK_TO_UNICODE[5095] := 16#5E0A;
   // GBK_TO_UNICODE[5096] := 16#8E8E;
   // GBK_TO_UNICODE[5097] := 16#5E0B;
   // GBK_TO_UNICODE[5098] := 16#8E8F;
   // GBK_TO_UNICODE[5099] := 16#5E0D;
   // GBK_TO_UNICODE[5100] := 16#8E90;
   // GBK_TO_UNICODE[5101] := 16#5E0E;
   // GBK_TO_UNICODE[5102] := 16#8E91;
   // GBK_TO_UNICODE[5103] := 16#5E12;
   // GBK_TO_UNICODE[5104] := 16#8E92;
   // GBK_TO_UNICODE[5105] := 16#5E13;
   // GBK_TO_UNICODE[5106] := 16#8E93;
   // GBK_TO_UNICODE[5107] := 16#5E17;
   // GBK_TO_UNICODE[5108] := 16#8E94;
   // GBK_TO_UNICODE[5109] := 16#5E1E;
   // GBK_TO_UNICODE[5110] := 16#8E95;
   // GBK_TO_UNICODE[5111] := 16#5E1F;
   // GBK_TO_UNICODE[5112] := 16#8E96;
   // GBK_TO_UNICODE[5113] := 16#5E20;
   // GBK_TO_UNICODE[5114] := 16#8E97;
   // GBK_TO_UNICODE[5115] := 16#5E21;
   // GBK_TO_UNICODE[5116] := 16#8E98;
   // GBK_TO_UNICODE[5117] := 16#5E22;
   // GBK_TO_UNICODE[5118] := 16#8E99;
   // GBK_TO_UNICODE[5119] := 16#5E23;
   // GBK_TO_UNICODE[5120] := 16#8E9A;
   // GBK_TO_UNICODE[5121] := 16#5E24;
   // GBK_TO_UNICODE[5122] := 16#8E9B;
   // GBK_TO_UNICODE[5123] := 16#5E25;
   // GBK_TO_UNICODE[5124] := 16#8E9C;
   // GBK_TO_UNICODE[5125] := 16#5E28;
   // GBK_TO_UNICODE[5126] := 16#8E9D;
   // GBK_TO_UNICODE[5127] := 16#5E29;
   // GBK_TO_UNICODE[5128] := 16#8E9E;
   // GBK_TO_UNICODE[5129] := 16#5E2A;
   // GBK_TO_UNICODE[5130] := 16#8E9F;
   // GBK_TO_UNICODE[5131] := 16#5E2B;
   // GBK_TO_UNICODE[5132] := 16#8EA0;
   // GBK_TO_UNICODE[5133] := 16#5E2C;
   // GBK_TO_UNICODE[5134] := 16#8EA1;
   // GBK_TO_UNICODE[5135] := 16#5E2F;
   // GBK_TO_UNICODE[5136] := 16#8EA2;
   // GBK_TO_UNICODE[5137] := 16#5E30;
   // GBK_TO_UNICODE[5138] := 16#8EA3;
   // GBK_TO_UNICODE[5139] := 16#5E32;
   // GBK_TO_UNICODE[5140] := 16#8EA4;
   // GBK_TO_UNICODE[5141] := 16#5E33;
   // GBK_TO_UNICODE[5142] := 16#8EA5;
   // GBK_TO_UNICODE[5143] := 16#5E34;
   // GBK_TO_UNICODE[5144] := 16#8EA6;
   // GBK_TO_UNICODE[5145] := 16#5E35;
   // GBK_TO_UNICODE[5146] := 16#8EA7;
   // GBK_TO_UNICODE[5147] := 16#5E36;
   // GBK_TO_UNICODE[5148] := 16#8EA8;
   // GBK_TO_UNICODE[5149] := 16#5E39;
   // GBK_TO_UNICODE[5150] := 16#8EA9;
   // GBK_TO_UNICODE[5151] := 16#5E3A;
   // GBK_TO_UNICODE[5152] := 16#8EAA;
   // GBK_TO_UNICODE[5153] := 16#5E3E;
   // GBK_TO_UNICODE[5154] := 16#8EAB;
   // GBK_TO_UNICODE[5155] := 16#5E3F;
   // GBK_TO_UNICODE[5156] := 16#8EAC;
   // GBK_TO_UNICODE[5157] := 16#5E40;
   // GBK_TO_UNICODE[5158] := 16#8EAD;
   // GBK_TO_UNICODE[5159] := 16#5E41;
   // GBK_TO_UNICODE[5160] := 16#8EAE;
   // GBK_TO_UNICODE[5161] := 16#5E43;
   // GBK_TO_UNICODE[5162] := 16#8EAF;
   // GBK_TO_UNICODE[5163] := 16#5E46;
   // GBK_TO_UNICODE[5164] := 16#8EB0;
   // GBK_TO_UNICODE[5165] := 16#5E47;
   // GBK_TO_UNICODE[5166] := 16#8EB1;
   // GBK_TO_UNICODE[5167] := 16#5E48;
   // GBK_TO_UNICODE[5168] := 16#8EB2;
   // GBK_TO_UNICODE[5169] := 16#5E49;
   // GBK_TO_UNICODE[5170] := 16#8EB3;
   // GBK_TO_UNICODE[5171] := 16#5E4A;
   // GBK_TO_UNICODE[5172] := 16#8EB4;
   // GBK_TO_UNICODE[5173] := 16#5E4B;
   // GBK_TO_UNICODE[5174] := 16#8EB5;
   // GBK_TO_UNICODE[5175] := 16#5E4D;
   // GBK_TO_UNICODE[5176] := 16#8EB6;
   // GBK_TO_UNICODE[5177] := 16#5E4E;
   // GBK_TO_UNICODE[5178] := 16#8EB7;
   // GBK_TO_UNICODE[5179] := 16#5E4F;
   // GBK_TO_UNICODE[5180] := 16#8EB8;
   // GBK_TO_UNICODE[5181] := 16#5E50;
   // GBK_TO_UNICODE[5182] := 16#8EB9;
   // GBK_TO_UNICODE[5183] := 16#5E51;
   // GBK_TO_UNICODE[5184] := 16#8EBA;
   // GBK_TO_UNICODE[5185] := 16#5E52;
   // GBK_TO_UNICODE[5186] := 16#8EBB;
   // GBK_TO_UNICODE[5187] := 16#5E53;
   // GBK_TO_UNICODE[5188] := 16#8EBC;
   // GBK_TO_UNICODE[5189] := 16#5E56;
   // GBK_TO_UNICODE[5190] := 16#8EBD;
   // GBK_TO_UNICODE[5191] := 16#5E57;
   // GBK_TO_UNICODE[5192] := 16#8EBE;
   // GBK_TO_UNICODE[5193] := 16#5E58;
   // GBK_TO_UNICODE[5194] := 16#8EBF;
   // GBK_TO_UNICODE[5195] := 16#5E59;
   // GBK_TO_UNICODE[5196] := 16#8EC0;
   // GBK_TO_UNICODE[5197] := 16#5E5A;
   // GBK_TO_UNICODE[5198] := 16#8EC1;
   // GBK_TO_UNICODE[5199] := 16#5E5C;
   // GBK_TO_UNICODE[5200] := 16#8EC2;
   // GBK_TO_UNICODE[5201] := 16#5E5D;
   // GBK_TO_UNICODE[5202] := 16#8EC3;
   // GBK_TO_UNICODE[5203] := 16#5E5F;
   // GBK_TO_UNICODE[5204] := 16#8EC4;
   // GBK_TO_UNICODE[5205] := 16#5E60;
   // GBK_TO_UNICODE[5206] := 16#8EC5;
   // GBK_TO_UNICODE[5207] := 16#5E63;
   // GBK_TO_UNICODE[5208] := 16#8EC6;
   // GBK_TO_UNICODE[5209] := 16#5E64;
   // GBK_TO_UNICODE[5210] := 16#8EC7;
   // GBK_TO_UNICODE[5211] := 16#5E65;
   // GBK_TO_UNICODE[5212] := 16#8EC8;
   // GBK_TO_UNICODE[5213] := 16#5E66;
   // GBK_TO_UNICODE[5214] := 16#8EC9;
   // GBK_TO_UNICODE[5215] := 16#5E67;
   // GBK_TO_UNICODE[5216] := 16#8ECA;
   // GBK_TO_UNICODE[5217] := 16#5E68;
   // GBK_TO_UNICODE[5218] := 16#8ECB;
   // GBK_TO_UNICODE[5219] := 16#5E69;
   // GBK_TO_UNICODE[5220] := 16#8ECC;
   // GBK_TO_UNICODE[5221] := 16#5E6A;
   // GBK_TO_UNICODE[5222] := 16#8ECD;
   // GBK_TO_UNICODE[5223] := 16#5E6B;
   // GBK_TO_UNICODE[5224] := 16#8ECE;
   // GBK_TO_UNICODE[5225] := 16#5E6C;
   // GBK_TO_UNICODE[5226] := 16#8ECF;
   // GBK_TO_UNICODE[5227] := 16#5E6D;
   // GBK_TO_UNICODE[5228] := 16#8ED0;
   // GBK_TO_UNICODE[5229] := 16#5E6E;
   // GBK_TO_UNICODE[5230] := 16#8ED1;
   // GBK_TO_UNICODE[5231] := 16#5E6F;
   // GBK_TO_UNICODE[5232] := 16#8ED2;
   // GBK_TO_UNICODE[5233] := 16#5E70;
   // GBK_TO_UNICODE[5234] := 16#8ED3;
   // GBK_TO_UNICODE[5235] := 16#5E71;
   // GBK_TO_UNICODE[5236] := 16#8ED4;
   // GBK_TO_UNICODE[5237] := 16#5E75;
   // GBK_TO_UNICODE[5238] := 16#8ED5;
   // GBK_TO_UNICODE[5239] := 16#5E77;
   // GBK_TO_UNICODE[5240] := 16#8ED6;
   // GBK_TO_UNICODE[5241] := 16#5E79;
   // GBK_TO_UNICODE[5242] := 16#8ED7;
   // GBK_TO_UNICODE[5243] := 16#5E7E;
   // GBK_TO_UNICODE[5244] := 16#8ED8;
   // GBK_TO_UNICODE[5245] := 16#5E81;
   // GBK_TO_UNICODE[5246] := 16#8ED9;
   // GBK_TO_UNICODE[5247] := 16#5E82;
   // GBK_TO_UNICODE[5248] := 16#8EDA;
   // GBK_TO_UNICODE[5249] := 16#5E83;
   // GBK_TO_UNICODE[5250] := 16#8EDB;
   // GBK_TO_UNICODE[5251] := 16#5E85;
   // GBK_TO_UNICODE[5252] := 16#8EDC;
   // GBK_TO_UNICODE[5253] := 16#5E88;
   // GBK_TO_UNICODE[5254] := 16#8EDD;
   // GBK_TO_UNICODE[5255] := 16#5E89;
   // GBK_TO_UNICODE[5256] := 16#8EDE;
   // GBK_TO_UNICODE[5257] := 16#5E8C;
   // GBK_TO_UNICODE[5258] := 16#8EDF;
   // GBK_TO_UNICODE[5259] := 16#5E8D;
   // GBK_TO_UNICODE[5260] := 16#8EE0;
   // GBK_TO_UNICODE[5261] := 16#5E8E;
   // GBK_TO_UNICODE[5262] := 16#8EE1;
   // GBK_TO_UNICODE[5263] := 16#5E92;
   // GBK_TO_UNICODE[5264] := 16#8EE2;
   // GBK_TO_UNICODE[5265] := 16#5E98;
   // GBK_TO_UNICODE[5266] := 16#8EE3;
   // GBK_TO_UNICODE[5267] := 16#5E9B;
   // GBK_TO_UNICODE[5268] := 16#8EE4;
   // GBK_TO_UNICODE[5269] := 16#5E9D;
   // GBK_TO_UNICODE[5270] := 16#8EE5;
   // GBK_TO_UNICODE[5271] := 16#5EA1;
   // GBK_TO_UNICODE[5272] := 16#8EE6;
   // GBK_TO_UNICODE[5273] := 16#5EA2;
   // GBK_TO_UNICODE[5274] := 16#8EE7;
   // GBK_TO_UNICODE[5275] := 16#5EA3;
   // GBK_TO_UNICODE[5276] := 16#8EE8;
   // GBK_TO_UNICODE[5277] := 16#5EA4;
   // GBK_TO_UNICODE[5278] := 16#8EE9;
   // GBK_TO_UNICODE[5279] := 16#5EA8;
   // GBK_TO_UNICODE[5280] := 16#8EEA;
   // GBK_TO_UNICODE[5281] := 16#5EA9;
   // GBK_TO_UNICODE[5282] := 16#8EEB;
   // GBK_TO_UNICODE[5283] := 16#5EAA;
   // GBK_TO_UNICODE[5284] := 16#8EEC;
   // GBK_TO_UNICODE[5285] := 16#5EAB;
   // GBK_TO_UNICODE[5286] := 16#8EED;
   // GBK_TO_UNICODE[5287] := 16#5EAC;
   // GBK_TO_UNICODE[5288] := 16#8EEE;
   // GBK_TO_UNICODE[5289] := 16#5EAE;
   // GBK_TO_UNICODE[5290] := 16#8EEF;
   // GBK_TO_UNICODE[5291] := 16#5EAF;
   // GBK_TO_UNICODE[5292] := 16#8EF0;
   // GBK_TO_UNICODE[5293] := 16#5EB0;
   // GBK_TO_UNICODE[5294] := 16#8EF1;
   // GBK_TO_UNICODE[5295] := 16#5EB1;
   // GBK_TO_UNICODE[5296] := 16#8EF2;
   // GBK_TO_UNICODE[5297] := 16#5EB2;
   // GBK_TO_UNICODE[5298] := 16#8EF3;
   // GBK_TO_UNICODE[5299] := 16#5EB4;
   // GBK_TO_UNICODE[5300] := 16#8EF4;
   // GBK_TO_UNICODE[5301] := 16#5EBA;
   // GBK_TO_UNICODE[5302] := 16#8EF5;
   // GBK_TO_UNICODE[5303] := 16#5EBB;
   // GBK_TO_UNICODE[5304] := 16#8EF6;
   // GBK_TO_UNICODE[5305] := 16#5EBC;
   // GBK_TO_UNICODE[5306] := 16#8EF7;
   // GBK_TO_UNICODE[5307] := 16#5EBD;
   // GBK_TO_UNICODE[5308] := 16#8EF8;
   // GBK_TO_UNICODE[5309] := 16#5EBF;
   // GBK_TO_UNICODE[5310] := 16#8EF9;
   // GBK_TO_UNICODE[5311] := 16#5EC0;
   // GBK_TO_UNICODE[5312] := 16#8EFA;
   // GBK_TO_UNICODE[5313] := 16#5EC1;
   // GBK_TO_UNICODE[5314] := 16#8EFB;
   // GBK_TO_UNICODE[5315] := 16#5EC2;
   // GBK_TO_UNICODE[5316] := 16#8EFC;
   // GBK_TO_UNICODE[5317] := 16#5EC3;
   // GBK_TO_UNICODE[5318] := 16#8EFD;
   // GBK_TO_UNICODE[5319] := 16#5EC4;
   // GBK_TO_UNICODE[5320] := 16#8EFE;
   // GBK_TO_UNICODE[5321] := 16#5EC5;
   // GBK_TO_UNICODE[5322] := 16#8F40;
   // GBK_TO_UNICODE[5323] := 16#5EC6;
   // GBK_TO_UNICODE[5324] := 16#8F41;
   // GBK_TO_UNICODE[5325] := 16#5EC7;
   // GBK_TO_UNICODE[5326] := 16#8F42;
   // GBK_TO_UNICODE[5327] := 16#5EC8;
   // GBK_TO_UNICODE[5328] := 16#8F43;
   // GBK_TO_UNICODE[5329] := 16#5ECB;
   // GBK_TO_UNICODE[5330] := 16#8F44;
   // GBK_TO_UNICODE[5331] := 16#5ECC;
   // GBK_TO_UNICODE[5332] := 16#8F45;
   // GBK_TO_UNICODE[5333] := 16#5ECD;
   // GBK_TO_UNICODE[5334] := 16#8F46;
   // GBK_TO_UNICODE[5335] := 16#5ECE;
   // GBK_TO_UNICODE[5336] := 16#8F47;
   // GBK_TO_UNICODE[5337] := 16#5ECF;
   // GBK_TO_UNICODE[5338] := 16#8F48;
   // GBK_TO_UNICODE[5339] := 16#5ED0;
   // GBK_TO_UNICODE[5340] := 16#8F49;
   // GBK_TO_UNICODE[5341] := 16#5ED4;
   // GBK_TO_UNICODE[5342] := 16#8F4A;
   // GBK_TO_UNICODE[5343] := 16#5ED5;
   // GBK_TO_UNICODE[5344] := 16#8F4B;
   // GBK_TO_UNICODE[5345] := 16#5ED7;
   // GBK_TO_UNICODE[5346] := 16#8F4C;
   // GBK_TO_UNICODE[5347] := 16#5ED8;
   // GBK_TO_UNICODE[5348] := 16#8F4D;
   // GBK_TO_UNICODE[5349] := 16#5ED9;
   // GBK_TO_UNICODE[5350] := 16#8F4E;
   // GBK_TO_UNICODE[5351] := 16#5EDA;
   // GBK_TO_UNICODE[5352] := 16#8F4F;
   // GBK_TO_UNICODE[5353] := 16#5EDC;
   // GBK_TO_UNICODE[5354] := 16#8F50;
   // GBK_TO_UNICODE[5355] := 16#5EDD;
   // GBK_TO_UNICODE[5356] := 16#8F51;
   // GBK_TO_UNICODE[5357] := 16#5EDE;
   // GBK_TO_UNICODE[5358] := 16#8F52;
   // GBK_TO_UNICODE[5359] := 16#5EDF;
   // GBK_TO_UNICODE[5360] := 16#8F53;
   // GBK_TO_UNICODE[5361] := 16#5EE0;
   // GBK_TO_UNICODE[5362] := 16#8F54;
   // GBK_TO_UNICODE[5363] := 16#5EE1;
   // GBK_TO_UNICODE[5364] := 16#8F55;
   // GBK_TO_UNICODE[5365] := 16#5EE2;
   // GBK_TO_UNICODE[5366] := 16#8F56;
   // GBK_TO_UNICODE[5367] := 16#5EE3;
   // GBK_TO_UNICODE[5368] := 16#8F57;
   // GBK_TO_UNICODE[5369] := 16#5EE4;
   // GBK_TO_UNICODE[5370] := 16#8F58;
   // GBK_TO_UNICODE[5371] := 16#5EE5;
   // GBK_TO_UNICODE[5372] := 16#8F59;
   // GBK_TO_UNICODE[5373] := 16#5EE6;
   // GBK_TO_UNICODE[5374] := 16#8F5A;
   // GBK_TO_UNICODE[5375] := 16#5EE7;
   // GBK_TO_UNICODE[5376] := 16#8F5B;
   // GBK_TO_UNICODE[5377] := 16#5EE9;
   // GBK_TO_UNICODE[5378] := 16#8F5C;
   // GBK_TO_UNICODE[5379] := 16#5EEB;
   // GBK_TO_UNICODE[5380] := 16#8F5D;
   // GBK_TO_UNICODE[5381] := 16#5EEC;
   // GBK_TO_UNICODE[5382] := 16#8F5E;
   // GBK_TO_UNICODE[5383] := 16#5EED;
   // GBK_TO_UNICODE[5384] := 16#8F5F;
   // GBK_TO_UNICODE[5385] := 16#5EEE;
   // GBK_TO_UNICODE[5386] := 16#8F60;
   // GBK_TO_UNICODE[5387] := 16#5EEF;
   // GBK_TO_UNICODE[5388] := 16#8F61;
   // GBK_TO_UNICODE[5389] := 16#5EF0;
   // GBK_TO_UNICODE[5390] := 16#8F62;
   // GBK_TO_UNICODE[5391] := 16#5EF1;
   // GBK_TO_UNICODE[5392] := 16#8F63;
   // GBK_TO_UNICODE[5393] := 16#5EF2;
   // GBK_TO_UNICODE[5394] := 16#8F64;
   // GBK_TO_UNICODE[5395] := 16#5EF3;
   // GBK_TO_UNICODE[5396] := 16#8F65;
   // GBK_TO_UNICODE[5397] := 16#5EF5;
   // GBK_TO_UNICODE[5398] := 16#8F66;
   // GBK_TO_UNICODE[5399] := 16#5EF8;
   // GBK_TO_UNICODE[5400] := 16#8F67;
   // GBK_TO_UNICODE[5401] := 16#5EF9;
   // GBK_TO_UNICODE[5402] := 16#8F68;
   // GBK_TO_UNICODE[5403] := 16#5EFB;
   // GBK_TO_UNICODE[5404] := 16#8F69;
   // GBK_TO_UNICODE[5405] := 16#5EFC;
   // GBK_TO_UNICODE[5406] := 16#8F6A;
   // GBK_TO_UNICODE[5407] := 16#5EFD;
   // GBK_TO_UNICODE[5408] := 16#8F6B;
   // GBK_TO_UNICODE[5409] := 16#5F05;
   // GBK_TO_UNICODE[5410] := 16#8F6C;
   // GBK_TO_UNICODE[5411] := 16#5F06;
   // GBK_TO_UNICODE[5412] := 16#8F6D;
   // GBK_TO_UNICODE[5413] := 16#5F07;
   // GBK_TO_UNICODE[5414] := 16#8F6E;
   // GBK_TO_UNICODE[5415] := 16#5F09;
   // GBK_TO_UNICODE[5416] := 16#8F6F;
   // GBK_TO_UNICODE[5417] := 16#5F0C;
   // GBK_TO_UNICODE[5418] := 16#8F70;
   // GBK_TO_UNICODE[5419] := 16#5F0D;
   // GBK_TO_UNICODE[5420] := 16#8F71;
   // GBK_TO_UNICODE[5421] := 16#5F0E;
   // GBK_TO_UNICODE[5422] := 16#8F72;
   // GBK_TO_UNICODE[5423] := 16#5F10;
   // GBK_TO_UNICODE[5424] := 16#8F73;
   // GBK_TO_UNICODE[5425] := 16#5F12;
   // GBK_TO_UNICODE[5426] := 16#8F74;
   // GBK_TO_UNICODE[5427] := 16#5F14;
   // GBK_TO_UNICODE[5428] := 16#8F75;
   // GBK_TO_UNICODE[5429] := 16#5F16;
   // GBK_TO_UNICODE[5430] := 16#8F76;
   // GBK_TO_UNICODE[5431] := 16#5F19;
   // GBK_TO_UNICODE[5432] := 16#8F77;
   // GBK_TO_UNICODE[5433] := 16#5F1A;
   // GBK_TO_UNICODE[5434] := 16#8F78;
   // GBK_TO_UNICODE[5435] := 16#5F1C;
   // GBK_TO_UNICODE[5436] := 16#8F79;
   // GBK_TO_UNICODE[5437] := 16#5F1D;
   // GBK_TO_UNICODE[5438] := 16#8F7A;
   // GBK_TO_UNICODE[5439] := 16#5F1E;
   // GBK_TO_UNICODE[5440] := 16#8F7B;
   // GBK_TO_UNICODE[5441] := 16#5F21;
   // GBK_TO_UNICODE[5442] := 16#8F7C;
   // GBK_TO_UNICODE[5443] := 16#5F22;
   // GBK_TO_UNICODE[5444] := 16#8F7D;
   // GBK_TO_UNICODE[5445] := 16#5F23;
   // GBK_TO_UNICODE[5446] := 16#8F7E;
   // GBK_TO_UNICODE[5447] := 16#5F24;
   // GBK_TO_UNICODE[5448] := 16#8F80;
   // GBK_TO_UNICODE[5449] := 16#5F28;
   // GBK_TO_UNICODE[5450] := 16#8F81;
   // GBK_TO_UNICODE[5451] := 16#5F2B;
   // GBK_TO_UNICODE[5452] := 16#8F82;
   // GBK_TO_UNICODE[5453] := 16#5F2C;
   // GBK_TO_UNICODE[5454] := 16#8F83;
   // GBK_TO_UNICODE[5455] := 16#5F2E;
   // GBK_TO_UNICODE[5456] := 16#8F84;
   // GBK_TO_UNICODE[5457] := 16#5F30;
   // GBK_TO_UNICODE[5458] := 16#8F85;
   // GBK_TO_UNICODE[5459] := 16#5F32;
   // GBK_TO_UNICODE[5460] := 16#8F86;
   // GBK_TO_UNICODE[5461] := 16#5F33;
   // GBK_TO_UNICODE[5462] := 16#8F87;
   // GBK_TO_UNICODE[5463] := 16#5F34;
   // GBK_TO_UNICODE[5464] := 16#8F88;
   // GBK_TO_UNICODE[5465] := 16#5F35;
   // GBK_TO_UNICODE[5466] := 16#8F89;
   // GBK_TO_UNICODE[5467] := 16#5F36;
   // GBK_TO_UNICODE[5468] := 16#8F8A;
   // GBK_TO_UNICODE[5469] := 16#5F37;
   // GBK_TO_UNICODE[5470] := 16#8F8B;
   // GBK_TO_UNICODE[5471] := 16#5F38;
   // GBK_TO_UNICODE[5472] := 16#8F8C;
   // GBK_TO_UNICODE[5473] := 16#5F3B;
   // GBK_TO_UNICODE[5474] := 16#8F8D;
   // GBK_TO_UNICODE[5475] := 16#5F3D;
   // GBK_TO_UNICODE[5476] := 16#8F8E;
   // GBK_TO_UNICODE[5477] := 16#5F3E;
   // GBK_TO_UNICODE[5478] := 16#8F8F;
   // GBK_TO_UNICODE[5479] := 16#5F3F;
   // GBK_TO_UNICODE[5480] := 16#8F90;
   // GBK_TO_UNICODE[5481] := 16#5F41;
   // GBK_TO_UNICODE[5482] := 16#8F91;
   // GBK_TO_UNICODE[5483] := 16#5F42;
   // GBK_TO_UNICODE[5484] := 16#8F92;
   // GBK_TO_UNICODE[5485] := 16#5F43;
   // GBK_TO_UNICODE[5486] := 16#8F93;
   // GBK_TO_UNICODE[5487] := 16#5F44;
   // GBK_TO_UNICODE[5488] := 16#8F94;
   // GBK_TO_UNICODE[5489] := 16#5F45;
   // GBK_TO_UNICODE[5490] := 16#8F95;
   // GBK_TO_UNICODE[5491] := 16#5F46;
   // GBK_TO_UNICODE[5492] := 16#8F96;
   // GBK_TO_UNICODE[5493] := 16#5F47;
   // GBK_TO_UNICODE[5494] := 16#8F97;
   // GBK_TO_UNICODE[5495] := 16#5F48;
   // GBK_TO_UNICODE[5496] := 16#8F98;
   // GBK_TO_UNICODE[5497] := 16#5F49;
   // GBK_TO_UNICODE[5498] := 16#8F99;
   // GBK_TO_UNICODE[5499] := 16#5F4A;
   // GBK_TO_UNICODE[5500] := 16#8F9A;
   // GBK_TO_UNICODE[5501] := 16#5F4B;
   // GBK_TO_UNICODE[5502] := 16#8F9B;
   // GBK_TO_UNICODE[5503] := 16#5F4C;
   // GBK_TO_UNICODE[5504] := 16#8F9C;
   // GBK_TO_UNICODE[5505] := 16#5F4D;
   // GBK_TO_UNICODE[5506] := 16#8F9D;
   // GBK_TO_UNICODE[5507] := 16#5F4E;
   // GBK_TO_UNICODE[5508] := 16#8F9E;
   // GBK_TO_UNICODE[5509] := 16#5F4F;
   // GBK_TO_UNICODE[5510] := 16#8F9F;
   // GBK_TO_UNICODE[5511] := 16#5F51;
   // GBK_TO_UNICODE[5512] := 16#8FA0;
   // GBK_TO_UNICODE[5513] := 16#5F54;
   // GBK_TO_UNICODE[5514] := 16#8FA1;
   // GBK_TO_UNICODE[5515] := 16#5F59;
   // GBK_TO_UNICODE[5516] := 16#8FA2;
   // GBK_TO_UNICODE[5517] := 16#5F5A;
   // GBK_TO_UNICODE[5518] := 16#8FA3;
   // GBK_TO_UNICODE[5519] := 16#5F5B;
   // GBK_TO_UNICODE[5520] := 16#8FA4;
   // GBK_TO_UNICODE[5521] := 16#5F5C;
   // GBK_TO_UNICODE[5522] := 16#8FA5;
   // GBK_TO_UNICODE[5523] := 16#5F5E;
   // GBK_TO_UNICODE[5524] := 16#8FA6;
   // GBK_TO_UNICODE[5525] := 16#5F5F;
   // GBK_TO_UNICODE[5526] := 16#8FA7;
   // GBK_TO_UNICODE[5527] := 16#5F60;
   // GBK_TO_UNICODE[5528] := 16#8FA8;
   // GBK_TO_UNICODE[5529] := 16#5F63;
   // GBK_TO_UNICODE[5530] := 16#8FA9;
   // GBK_TO_UNICODE[5531] := 16#5F65;
   // GBK_TO_UNICODE[5532] := 16#8FAA;
   // GBK_TO_UNICODE[5533] := 16#5F67;
   // GBK_TO_UNICODE[5534] := 16#8FAB;
   // GBK_TO_UNICODE[5535] := 16#5F68;
   // GBK_TO_UNICODE[5536] := 16#8FAC;
   // GBK_TO_UNICODE[5537] := 16#5F6B;
   // GBK_TO_UNICODE[5538] := 16#8FAD;
   // GBK_TO_UNICODE[5539] := 16#5F6E;
   // GBK_TO_UNICODE[5540] := 16#8FAE;
   // GBK_TO_UNICODE[5541] := 16#5F6F;
   // GBK_TO_UNICODE[5542] := 16#8FAF;
   // GBK_TO_UNICODE[5543] := 16#5F72;
   // GBK_TO_UNICODE[5544] := 16#8FB0;
   // GBK_TO_UNICODE[5545] := 16#5F74;
   // GBK_TO_UNICODE[5546] := 16#8FB1;
   // GBK_TO_UNICODE[5547] := 16#5F75;
   // GBK_TO_UNICODE[5548] := 16#8FB2;
   // GBK_TO_UNICODE[5549] := 16#5F76;
   // GBK_TO_UNICODE[5550] := 16#8FB3;
   // GBK_TO_UNICODE[5551] := 16#5F78;
   // GBK_TO_UNICODE[5552] := 16#8FB4;
   // GBK_TO_UNICODE[5553] := 16#5F7A;
   // GBK_TO_UNICODE[5554] := 16#8FB5;
   // GBK_TO_UNICODE[5555] := 16#5F7D;
   // GBK_TO_UNICODE[5556] := 16#8FB6;
   // GBK_TO_UNICODE[5557] := 16#5F7E;
   // GBK_TO_UNICODE[5558] := 16#8FB7;
   // GBK_TO_UNICODE[5559] := 16#5F7F;
   // GBK_TO_UNICODE[5560] := 16#8FB8;
   // GBK_TO_UNICODE[5561] := 16#5F83;
   // GBK_TO_UNICODE[5562] := 16#8FB9;
   // GBK_TO_UNICODE[5563] := 16#5F86;
   // GBK_TO_UNICODE[5564] := 16#8FBA;
   // GBK_TO_UNICODE[5565] := 16#5F8D;
   // GBK_TO_UNICODE[5566] := 16#8FBB;
   // GBK_TO_UNICODE[5567] := 16#5F8E;
   // GBK_TO_UNICODE[5568] := 16#8FBC;
   // GBK_TO_UNICODE[5569] := 16#5F8F;
   // GBK_TO_UNICODE[5570] := 16#8FBD;
   // GBK_TO_UNICODE[5571] := 16#5F91;
   // GBK_TO_UNICODE[5572] := 16#8FBE;
   // GBK_TO_UNICODE[5573] := 16#5F93;
   // GBK_TO_UNICODE[5574] := 16#8FBF;
   // GBK_TO_UNICODE[5575] := 16#5F94;
   // GBK_TO_UNICODE[5576] := 16#8FC0;
   // GBK_TO_UNICODE[5577] := 16#5F96;
   // GBK_TO_UNICODE[5578] := 16#8FC1;
   // GBK_TO_UNICODE[5579] := 16#5F9A;
   // GBK_TO_UNICODE[5580] := 16#8FC2;
   // GBK_TO_UNICODE[5581] := 16#5F9B;
   // GBK_TO_UNICODE[5582] := 16#8FC3;
   // GBK_TO_UNICODE[5583] := 16#5F9D;
   // GBK_TO_UNICODE[5584] := 16#8FC4;
   // GBK_TO_UNICODE[5585] := 16#5F9E;
   // GBK_TO_UNICODE[5586] := 16#8FC5;
   // GBK_TO_UNICODE[5587] := 16#5F9F;
   // GBK_TO_UNICODE[5588] := 16#8FC6;
   // GBK_TO_UNICODE[5589] := 16#5FA0;
   // GBK_TO_UNICODE[5590] := 16#8FC7;
   // GBK_TO_UNICODE[5591] := 16#5FA2;
   // GBK_TO_UNICODE[5592] := 16#8FC8;
   // GBK_TO_UNICODE[5593] := 16#5FA3;
   // GBK_TO_UNICODE[5594] := 16#8FC9;
   // GBK_TO_UNICODE[5595] := 16#5FA4;
   // GBK_TO_UNICODE[5596] := 16#8FCA;
   // GBK_TO_UNICODE[5597] := 16#5FA5;
   // GBK_TO_UNICODE[5598] := 16#8FCB;
   // GBK_TO_UNICODE[5599] := 16#5FA6;
   // GBK_TO_UNICODE[5600] := 16#8FCC;
   // GBK_TO_UNICODE[5601] := 16#5FA7;
   // GBK_TO_UNICODE[5602] := 16#8FCD;
   // GBK_TO_UNICODE[5603] := 16#5FA9;
   // GBK_TO_UNICODE[5604] := 16#8FCE;
   // GBK_TO_UNICODE[5605] := 16#5FAB;
   // GBK_TO_UNICODE[5606] := 16#8FCF;
   // GBK_TO_UNICODE[5607] := 16#5FAC;
   // GBK_TO_UNICODE[5608] := 16#8FD0;
   // GBK_TO_UNICODE[5609] := 16#5FAF;
   // GBK_TO_UNICODE[5610] := 16#8FD1;
   // GBK_TO_UNICODE[5611] := 16#5FB0;
   // GBK_TO_UNICODE[5612] := 16#8FD2;
   // GBK_TO_UNICODE[5613] := 16#5FB1;
   // GBK_TO_UNICODE[5614] := 16#8FD3;
   // GBK_TO_UNICODE[5615] := 16#5FB2;
   // GBK_TO_UNICODE[5616] := 16#8FD4;
   // GBK_TO_UNICODE[5617] := 16#5FB3;
   // GBK_TO_UNICODE[5618] := 16#8FD5;
   // GBK_TO_UNICODE[5619] := 16#5FB4;
   // GBK_TO_UNICODE[5620] := 16#8FD6;
   // GBK_TO_UNICODE[5621] := 16#5FB6;
   // GBK_TO_UNICODE[5622] := 16#8FD7;
   // GBK_TO_UNICODE[5623] := 16#5FB8;
   // GBK_TO_UNICODE[5624] := 16#8FD8;
   // GBK_TO_UNICODE[5625] := 16#5FB9;
   // GBK_TO_UNICODE[5626] := 16#8FD9;
   // GBK_TO_UNICODE[5627] := 16#5FBA;
   // GBK_TO_UNICODE[5628] := 16#8FDA;
   // GBK_TO_UNICODE[5629] := 16#5FBB;
   // GBK_TO_UNICODE[5630] := 16#8FDB;
   // GBK_TO_UNICODE[5631] := 16#5FBE;
   // GBK_TO_UNICODE[5632] := 16#8FDC;
   // GBK_TO_UNICODE[5633] := 16#5FBF;
   // GBK_TO_UNICODE[5634] := 16#8FDD;
   // GBK_TO_UNICODE[5635] := 16#5FC0;
   // GBK_TO_UNICODE[5636] := 16#8FDE;
   // GBK_TO_UNICODE[5637] := 16#5FC1;
   // GBK_TO_UNICODE[5638] := 16#8FDF;
   // GBK_TO_UNICODE[5639] := 16#5FC2;
   // GBK_TO_UNICODE[5640] := 16#8FE0;
   // GBK_TO_UNICODE[5641] := 16#5FC7;
   // GBK_TO_UNICODE[5642] := 16#8FE1;
   // GBK_TO_UNICODE[5643] := 16#5FC8;
   // GBK_TO_UNICODE[5644] := 16#8FE2;
   // GBK_TO_UNICODE[5645] := 16#5FCA;
   // GBK_TO_UNICODE[5646] := 16#8FE3;
   // GBK_TO_UNICODE[5647] := 16#5FCB;
   // GBK_TO_UNICODE[5648] := 16#8FE4;
   // GBK_TO_UNICODE[5649] := 16#5FCE;
   // GBK_TO_UNICODE[5650] := 16#8FE5;
   // GBK_TO_UNICODE[5651] := 16#5FD3;
   // GBK_TO_UNICODE[5652] := 16#8FE6;
   // GBK_TO_UNICODE[5653] := 16#5FD4;
   // GBK_TO_UNICODE[5654] := 16#8FE7;
   // GBK_TO_UNICODE[5655] := 16#5FD5;
   // GBK_TO_UNICODE[5656] := 16#8FE8;
   // GBK_TO_UNICODE[5657] := 16#5FDA;
   // GBK_TO_UNICODE[5658] := 16#8FE9;
   // GBK_TO_UNICODE[5659] := 16#5FDB;
   // GBK_TO_UNICODE[5660] := 16#8FEA;
   // GBK_TO_UNICODE[5661] := 16#5FDC;
   // GBK_TO_UNICODE[5662] := 16#8FEB;
   // GBK_TO_UNICODE[5663] := 16#5FDE;
   // GBK_TO_UNICODE[5664] := 16#8FEC;
   // GBK_TO_UNICODE[5665] := 16#5FDF;
   // GBK_TO_UNICODE[5666] := 16#8FED;
   // GBK_TO_UNICODE[5667] := 16#5FE2;
   // GBK_TO_UNICODE[5668] := 16#8FEE;
   // GBK_TO_UNICODE[5669] := 16#5FE3;
   // GBK_TO_UNICODE[5670] := 16#8FEF;
   // GBK_TO_UNICODE[5671] := 16#5FE5;
   // GBK_TO_UNICODE[5672] := 16#8FF0;
   // GBK_TO_UNICODE[5673] := 16#5FE6;
   // GBK_TO_UNICODE[5674] := 16#8FF1;
   // GBK_TO_UNICODE[5675] := 16#5FE8;
   // GBK_TO_UNICODE[5676] := 16#8FF2;
   // GBK_TO_UNICODE[5677] := 16#5FE9;
   // GBK_TO_UNICODE[5678] := 16#8FF3;
   // GBK_TO_UNICODE[5679] := 16#5FEC;
   // GBK_TO_UNICODE[5680] := 16#8FF4;
   // GBK_TO_UNICODE[5681] := 16#5FEF;
   // GBK_TO_UNICODE[5682] := 16#8FF5;
   // GBK_TO_UNICODE[5683] := 16#5FF0;
   // GBK_TO_UNICODE[5684] := 16#8FF6;
   // GBK_TO_UNICODE[5685] := 16#5FF2;
   // GBK_TO_UNICODE[5686] := 16#8FF7;
   // GBK_TO_UNICODE[5687] := 16#5FF3;
   // GBK_TO_UNICODE[5688] := 16#8FF8;
   // GBK_TO_UNICODE[5689] := 16#5FF4;
   // GBK_TO_UNICODE[5690] := 16#8FF9;
   // GBK_TO_UNICODE[5691] := 16#5FF6;
   // GBK_TO_UNICODE[5692] := 16#8FFA;
   // GBK_TO_UNICODE[5693] := 16#5FF7;
   // GBK_TO_UNICODE[5694] := 16#8FFB;
   // GBK_TO_UNICODE[5695] := 16#5FF9;
   // GBK_TO_UNICODE[5696] := 16#8FFC;
   // GBK_TO_UNICODE[5697] := 16#5FFA;
   // GBK_TO_UNICODE[5698] := 16#8FFD;
   // GBK_TO_UNICODE[5699] := 16#5FFC;
   // GBK_TO_UNICODE[5700] := 16#8FFE;
   // GBK_TO_UNICODE[5701] := 16#6007;
   // GBK_TO_UNICODE[5702] := 16#9040;
   // GBK_TO_UNICODE[5703] := 16#6008;
   // GBK_TO_UNICODE[5704] := 16#9041;
   // GBK_TO_UNICODE[5705] := 16#6009;
   // GBK_TO_UNICODE[5706] := 16#9042;
   // GBK_TO_UNICODE[5707] := 16#600B;
   // GBK_TO_UNICODE[5708] := 16#9043;
   // GBK_TO_UNICODE[5709] := 16#600C;
   // GBK_TO_UNICODE[5710] := 16#9044;
   // GBK_TO_UNICODE[5711] := 16#6010;
   // GBK_TO_UNICODE[5712] := 16#9045;
   // GBK_TO_UNICODE[5713] := 16#6011;
   // GBK_TO_UNICODE[5714] := 16#9046;
   // GBK_TO_UNICODE[5715] := 16#6013;
   // GBK_TO_UNICODE[5716] := 16#9047;
   // GBK_TO_UNICODE[5717] := 16#6017;
   // GBK_TO_UNICODE[5718] := 16#9048;
   // GBK_TO_UNICODE[5719] := 16#6018;
   // GBK_TO_UNICODE[5720] := 16#9049;
   // GBK_TO_UNICODE[5721] := 16#601A;
   // GBK_TO_UNICODE[5722] := 16#904A;
   // GBK_TO_UNICODE[5723] := 16#601E;
   // GBK_TO_UNICODE[5724] := 16#904B;
   // GBK_TO_UNICODE[5725] := 16#601F;
   // GBK_TO_UNICODE[5726] := 16#904C;
   // GBK_TO_UNICODE[5727] := 16#6022;
   // GBK_TO_UNICODE[5728] := 16#904D;
   // GBK_TO_UNICODE[5729] := 16#6023;
   // GBK_TO_UNICODE[5730] := 16#904E;
   // GBK_TO_UNICODE[5731] := 16#6024;
   // GBK_TO_UNICODE[5732] := 16#904F;
   // GBK_TO_UNICODE[5733] := 16#602C;
   // GBK_TO_UNICODE[5734] := 16#9050;
   // GBK_TO_UNICODE[5735] := 16#602D;
   // GBK_TO_UNICODE[5736] := 16#9051;
   // GBK_TO_UNICODE[5737] := 16#602E;
   // GBK_TO_UNICODE[5738] := 16#9052;
   // GBK_TO_UNICODE[5739] := 16#6030;
   // GBK_TO_UNICODE[5740] := 16#9053;
   // GBK_TO_UNICODE[5741] := 16#6031;
   // GBK_TO_UNICODE[5742] := 16#9054;
   // GBK_TO_UNICODE[5743] := 16#6032;
   // GBK_TO_UNICODE[5744] := 16#9055;
   // GBK_TO_UNICODE[5745] := 16#6033;
   // GBK_TO_UNICODE[5746] := 16#9056;
   // GBK_TO_UNICODE[5747] := 16#6034;
   // GBK_TO_UNICODE[5748] := 16#9057;
   // GBK_TO_UNICODE[5749] := 16#6036;
   // GBK_TO_UNICODE[5750] := 16#9058;
   // GBK_TO_UNICODE[5751] := 16#6037;
   // GBK_TO_UNICODE[5752] := 16#9059;
   // GBK_TO_UNICODE[5753] := 16#6038;
   // GBK_TO_UNICODE[5754] := 16#905A;
   // GBK_TO_UNICODE[5755] := 16#6039;
   // GBK_TO_UNICODE[5756] := 16#905B;
   // GBK_TO_UNICODE[5757] := 16#603A;
   // GBK_TO_UNICODE[5758] := 16#905C;
   // GBK_TO_UNICODE[5759] := 16#603D;
   // GBK_TO_UNICODE[5760] := 16#905D;
   // GBK_TO_UNICODE[5761] := 16#603E;
   // GBK_TO_UNICODE[5762] := 16#905E;
   // GBK_TO_UNICODE[5763] := 16#6040;
   // GBK_TO_UNICODE[5764] := 16#905F;
   // GBK_TO_UNICODE[5765] := 16#6044;
   // GBK_TO_UNICODE[5766] := 16#9060;
   // GBK_TO_UNICODE[5767] := 16#6045;
   // GBK_TO_UNICODE[5768] := 16#9061;
   // GBK_TO_UNICODE[5769] := 16#6046;
   // GBK_TO_UNICODE[5770] := 16#9062;
   // GBK_TO_UNICODE[5771] := 16#6047;
   // GBK_TO_UNICODE[5772] := 16#9063;
   // GBK_TO_UNICODE[5773] := 16#6048;
   // GBK_TO_UNICODE[5774] := 16#9064;
   // GBK_TO_UNICODE[5775] := 16#6049;
   // GBK_TO_UNICODE[5776] := 16#9065;
   // GBK_TO_UNICODE[5777] := 16#604A;
   // GBK_TO_UNICODE[5778] := 16#9066;
   // GBK_TO_UNICODE[5779] := 16#604C;
   // GBK_TO_UNICODE[5780] := 16#9067;
   // GBK_TO_UNICODE[5781] := 16#604E;
   // GBK_TO_UNICODE[5782] := 16#9068;
   // GBK_TO_UNICODE[5783] := 16#604F;
   // GBK_TO_UNICODE[5784] := 16#9069;
   // GBK_TO_UNICODE[5785] := 16#6051;
   // GBK_TO_UNICODE[5786] := 16#906A;
   // GBK_TO_UNICODE[5787] := 16#6053;
   // GBK_TO_UNICODE[5788] := 16#906B;
   // GBK_TO_UNICODE[5789] := 16#6054;
   // GBK_TO_UNICODE[5790] := 16#906C;
   // GBK_TO_UNICODE[5791] := 16#6056;
   // GBK_TO_UNICODE[5792] := 16#906D;
   // GBK_TO_UNICODE[5793] := 16#6057;
   // GBK_TO_UNICODE[5794] := 16#906E;
   // GBK_TO_UNICODE[5795] := 16#6058;
   // GBK_TO_UNICODE[5796] := 16#906F;
   // GBK_TO_UNICODE[5797] := 16#605B;
   // GBK_TO_UNICODE[5798] := 16#9070;
   // GBK_TO_UNICODE[5799] := 16#605C;
   // GBK_TO_UNICODE[5800] := 16#9071;
   // GBK_TO_UNICODE[5801] := 16#605E;
   // GBK_TO_UNICODE[5802] := 16#9072;
   // GBK_TO_UNICODE[5803] := 16#605F;
   // GBK_TO_UNICODE[5804] := 16#9073;
   // GBK_TO_UNICODE[5805] := 16#6060;
   // GBK_TO_UNICODE[5806] := 16#9074;
   // GBK_TO_UNICODE[5807] := 16#6061;
   // GBK_TO_UNICODE[5808] := 16#9075;
   // GBK_TO_UNICODE[5809] := 16#6065;
   // GBK_TO_UNICODE[5810] := 16#9076;
   // GBK_TO_UNICODE[5811] := 16#6066;
   // GBK_TO_UNICODE[5812] := 16#9077;
   // GBK_TO_UNICODE[5813] := 16#606E;
   // GBK_TO_UNICODE[5814] := 16#9078;
   // GBK_TO_UNICODE[5815] := 16#6071;
   // GBK_TO_UNICODE[5816] := 16#9079;
   // GBK_TO_UNICODE[5817] := 16#6072;
   // GBK_TO_UNICODE[5818] := 16#907A;
   // GBK_TO_UNICODE[5819] := 16#6074;
   // GBK_TO_UNICODE[5820] := 16#907B;
   // GBK_TO_UNICODE[5821] := 16#6075;
   // GBK_TO_UNICODE[5822] := 16#907C;
   // GBK_TO_UNICODE[5823] := 16#6077;
   // GBK_TO_UNICODE[5824] := 16#907D;
   // GBK_TO_UNICODE[5825] := 16#607E;
   // GBK_TO_UNICODE[5826] := 16#907E;
   // GBK_TO_UNICODE[5827] := 16#6080;
   // GBK_TO_UNICODE[5828] := 16#9080;
   // GBK_TO_UNICODE[5829] := 16#6081;
   // GBK_TO_UNICODE[5830] := 16#9081;
   // GBK_TO_UNICODE[5831] := 16#6082;
   // GBK_TO_UNICODE[5832] := 16#9082;
   // GBK_TO_UNICODE[5833] := 16#6085;
   // GBK_TO_UNICODE[5834] := 16#9083;
   // GBK_TO_UNICODE[5835] := 16#6086;
   // GBK_TO_UNICODE[5836] := 16#9084;
   // GBK_TO_UNICODE[5837] := 16#6087;
   // GBK_TO_UNICODE[5838] := 16#9085;
   // GBK_TO_UNICODE[5839] := 16#6088;
   // GBK_TO_UNICODE[5840] := 16#9086;
   // GBK_TO_UNICODE[5841] := 16#608A;
   // GBK_TO_UNICODE[5842] := 16#9087;
   // GBK_TO_UNICODE[5843] := 16#608B;
   // GBK_TO_UNICODE[5844] := 16#9088;
   // GBK_TO_UNICODE[5845] := 16#608E;
   // GBK_TO_UNICODE[5846] := 16#9089;
   // GBK_TO_UNICODE[5847] := 16#608F;
   // GBK_TO_UNICODE[5848] := 16#908A;
   // GBK_TO_UNICODE[5849] := 16#6090;
   // GBK_TO_UNICODE[5850] := 16#908B;
   // GBK_TO_UNICODE[5851] := 16#6091;
   // GBK_TO_UNICODE[5852] := 16#908C;
   // GBK_TO_UNICODE[5853] := 16#6093;
   // GBK_TO_UNICODE[5854] := 16#908D;
   // GBK_TO_UNICODE[5855] := 16#6095;
   // GBK_TO_UNICODE[5856] := 16#908E;
   // GBK_TO_UNICODE[5857] := 16#6097;
   // GBK_TO_UNICODE[5858] := 16#908F;
   // GBK_TO_UNICODE[5859] := 16#6098;
   // GBK_TO_UNICODE[5860] := 16#9090;
   // GBK_TO_UNICODE[5861] := 16#6099;
   // GBK_TO_UNICODE[5862] := 16#9091;
   // GBK_TO_UNICODE[5863] := 16#609C;
   // GBK_TO_UNICODE[5864] := 16#9092;
   // GBK_TO_UNICODE[5865] := 16#609E;
   // GBK_TO_UNICODE[5866] := 16#9093;
   // GBK_TO_UNICODE[5867] := 16#60A1;
   // GBK_TO_UNICODE[5868] := 16#9094;
   // GBK_TO_UNICODE[5869] := 16#60A2;
   // GBK_TO_UNICODE[5870] := 16#9095;
   // GBK_TO_UNICODE[5871] := 16#60A4;
   // GBK_TO_UNICODE[5872] := 16#9096;
   // GBK_TO_UNICODE[5873] := 16#60A5;
   // GBK_TO_UNICODE[5874] := 16#9097;
   // GBK_TO_UNICODE[5875] := 16#60A7;
   // GBK_TO_UNICODE[5876] := 16#9098;
   // GBK_TO_UNICODE[5877] := 16#60A9;
   // GBK_TO_UNICODE[5878] := 16#9099;
   // GBK_TO_UNICODE[5879] := 16#60AA;
   // GBK_TO_UNICODE[5880] := 16#909A;
   // GBK_TO_UNICODE[5881] := 16#60AE;
   // GBK_TO_UNICODE[5882] := 16#909B;
   // GBK_TO_UNICODE[5883] := 16#60B0;
   // GBK_TO_UNICODE[5884] := 16#909C;
   // GBK_TO_UNICODE[5885] := 16#60B3;
   // GBK_TO_UNICODE[5886] := 16#909D;
   // GBK_TO_UNICODE[5887] := 16#60B5;
   // GBK_TO_UNICODE[5888] := 16#909E;
   // GBK_TO_UNICODE[5889] := 16#60B6;
   // GBK_TO_UNICODE[5890] := 16#909F;
   // GBK_TO_UNICODE[5891] := 16#60B7;
   // GBK_TO_UNICODE[5892] := 16#90A0;
   // GBK_TO_UNICODE[5893] := 16#60B9;
   // GBK_TO_UNICODE[5894] := 16#90A1;
   // GBK_TO_UNICODE[5895] := 16#60BA;
   // GBK_TO_UNICODE[5896] := 16#90A2;
   // GBK_TO_UNICODE[5897] := 16#60BD;
   // GBK_TO_UNICODE[5898] := 16#90A3;
   // GBK_TO_UNICODE[5899] := 16#60BE;
   // GBK_TO_UNICODE[5900] := 16#90A4;
   // GBK_TO_UNICODE[5901] := 16#60BF;
   // GBK_TO_UNICODE[5902] := 16#90A5;
   // GBK_TO_UNICODE[5903] := 16#60C0;
   // GBK_TO_UNICODE[5904] := 16#90A6;
   // GBK_TO_UNICODE[5905] := 16#60C1;
   // GBK_TO_UNICODE[5906] := 16#90A7;
   // GBK_TO_UNICODE[5907] := 16#60C2;
   // GBK_TO_UNICODE[5908] := 16#90A8;
   // GBK_TO_UNICODE[5909] := 16#60C3;
   // GBK_TO_UNICODE[5910] := 16#90A9;
   // GBK_TO_UNICODE[5911] := 16#60C4;
   // GBK_TO_UNICODE[5912] := 16#90AA;
   // GBK_TO_UNICODE[5913] := 16#60C7;
   // GBK_TO_UNICODE[5914] := 16#90AB;
   // GBK_TO_UNICODE[5915] := 16#60C8;
   // GBK_TO_UNICODE[5916] := 16#90AC;
   // GBK_TO_UNICODE[5917] := 16#60C9;
   // GBK_TO_UNICODE[5918] := 16#90AD;
   // GBK_TO_UNICODE[5919] := 16#60CC;
   // GBK_TO_UNICODE[5920] := 16#90AE;
   // GBK_TO_UNICODE[5921] := 16#60CD;
   // GBK_TO_UNICODE[5922] := 16#90AF;
   // GBK_TO_UNICODE[5923] := 16#60CE;
   // GBK_TO_UNICODE[5924] := 16#90B0;
   // GBK_TO_UNICODE[5925] := 16#60CF;
   // GBK_TO_UNICODE[5926] := 16#90B1;
   // GBK_TO_UNICODE[5927] := 16#60D0;
   // GBK_TO_UNICODE[5928] := 16#90B2;
   // GBK_TO_UNICODE[5929] := 16#60D2;
   // GBK_TO_UNICODE[5930] := 16#90B3;
   // GBK_TO_UNICODE[5931] := 16#60D3;
   // GBK_TO_UNICODE[5932] := 16#90B4;
   // GBK_TO_UNICODE[5933] := 16#60D4;
   // GBK_TO_UNICODE[5934] := 16#90B5;
   // GBK_TO_UNICODE[5935] := 16#60D6;
   // GBK_TO_UNICODE[5936] := 16#90B6;
   // GBK_TO_UNICODE[5937] := 16#60D7;
   // GBK_TO_UNICODE[5938] := 16#90B7;
   // GBK_TO_UNICODE[5939] := 16#60D9;
   // GBK_TO_UNICODE[5940] := 16#90B8;
   // GBK_TO_UNICODE[5941] := 16#60DB;
   // GBK_TO_UNICODE[5942] := 16#90B9;
   // GBK_TO_UNICODE[5943] := 16#60DE;
   // GBK_TO_UNICODE[5944] := 16#90BA;
   // GBK_TO_UNICODE[5945] := 16#60E1;
   // GBK_TO_UNICODE[5946] := 16#90BB;
   // GBK_TO_UNICODE[5947] := 16#60E2;
   // GBK_TO_UNICODE[5948] := 16#90BC;
   // GBK_TO_UNICODE[5949] := 16#60E3;
   // GBK_TO_UNICODE[5950] := 16#90BD;
   // GBK_TO_UNICODE[5951] := 16#60E4;
   // GBK_TO_UNICODE[5952] := 16#90BE;
   // GBK_TO_UNICODE[5953] := 16#60E5;
   // GBK_TO_UNICODE[5954] := 16#90BF;
   // GBK_TO_UNICODE[5955] := 16#60EA;
   // GBK_TO_UNICODE[5956] := 16#90C0;
   // GBK_TO_UNICODE[5957] := 16#60F1;
   // GBK_TO_UNICODE[5958] := 16#90C1;
   // GBK_TO_UNICODE[5959] := 16#60F2;
   // GBK_TO_UNICODE[5960] := 16#90C2;
   // GBK_TO_UNICODE[5961] := 16#60F5;
   // GBK_TO_UNICODE[5962] := 16#90C3;
   // GBK_TO_UNICODE[5963] := 16#60F7;
   // GBK_TO_UNICODE[5964] := 16#90C4;
   // GBK_TO_UNICODE[5965] := 16#60F8;
   // GBK_TO_UNICODE[5966] := 16#90C5;
   // GBK_TO_UNICODE[5967] := 16#60FB;
   // GBK_TO_UNICODE[5968] := 16#90C6;
   // GBK_TO_UNICODE[5969] := 16#60FC;
   // GBK_TO_UNICODE[5970] := 16#90C7;
   // GBK_TO_UNICODE[5971] := 16#60FD;
   // GBK_TO_UNICODE[5972] := 16#90C8;
   // GBK_TO_UNICODE[5973] := 16#60FE;
   // GBK_TO_UNICODE[5974] := 16#90C9;
   // GBK_TO_UNICODE[5975] := 16#60FF;
   // GBK_TO_UNICODE[5976] := 16#90CA;
   // GBK_TO_UNICODE[5977] := 16#6102;
   // GBK_TO_UNICODE[5978] := 16#90CB;
   // GBK_TO_UNICODE[5979] := 16#6103;
   // GBK_TO_UNICODE[5980] := 16#90CC;
   // GBK_TO_UNICODE[5981] := 16#6104;
   // GBK_TO_UNICODE[5982] := 16#90CD;
   // GBK_TO_UNICODE[5983] := 16#6105;
   // GBK_TO_UNICODE[5984] := 16#90CE;
   // GBK_TO_UNICODE[5985] := 16#6107;
   // GBK_TO_UNICODE[5986] := 16#90CF;
   // GBK_TO_UNICODE[5987] := 16#610A;
   // GBK_TO_UNICODE[5988] := 16#90D0;
   // GBK_TO_UNICODE[5989] := 16#610B;
   // GBK_TO_UNICODE[5990] := 16#90D1;
   // GBK_TO_UNICODE[5991] := 16#610C;
   // GBK_TO_UNICODE[5992] := 16#90D2;
   // GBK_TO_UNICODE[5993] := 16#6110;
   // GBK_TO_UNICODE[5994] := 16#90D3;
   // GBK_TO_UNICODE[5995] := 16#6111;
   // GBK_TO_UNICODE[5996] := 16#90D4;
   // GBK_TO_UNICODE[5997] := 16#6112;
   // GBK_TO_UNICODE[5998] := 16#90D5;
   // GBK_TO_UNICODE[5999] := 16#6113;
   // GBK_TO_UNICODE[6000] := 16#90D6;
   // GBK_TO_UNICODE[6001] := 16#6114;
   // GBK_TO_UNICODE[6002] := 16#90D7;
   // GBK_TO_UNICODE[6003] := 16#6116;
   // GBK_TO_UNICODE[6004] := 16#90D8;
   // GBK_TO_UNICODE[6005] := 16#6117;
   // GBK_TO_UNICODE[6006] := 16#90D9;
   // GBK_TO_UNICODE[6007] := 16#6118;
   // GBK_TO_UNICODE[6008] := 16#90DA;
   // GBK_TO_UNICODE[6009] := 16#6119;
   // GBK_TO_UNICODE[6010] := 16#90DB;
   // GBK_TO_UNICODE[6011] := 16#611B;
   // GBK_TO_UNICODE[6012] := 16#90DC;
   // GBK_TO_UNICODE[6013] := 16#611C;
   // GBK_TO_UNICODE[6014] := 16#90DD;
   // GBK_TO_UNICODE[6015] := 16#611D;
   // GBK_TO_UNICODE[6016] := 16#90DE;
   // GBK_TO_UNICODE[6017] := 16#611E;
   // GBK_TO_UNICODE[6018] := 16#90DF;
   // GBK_TO_UNICODE[6019] := 16#6121;
   // GBK_TO_UNICODE[6020] := 16#90E0;
   // GBK_TO_UNICODE[6021] := 16#6122;
   // GBK_TO_UNICODE[6022] := 16#90E1;
   // GBK_TO_UNICODE[6023] := 16#6125;
   // GBK_TO_UNICODE[6024] := 16#90E2;
   // GBK_TO_UNICODE[6025] := 16#6128;
   // GBK_TO_UNICODE[6026] := 16#90E3;
   // GBK_TO_UNICODE[6027] := 16#6129;
   // GBK_TO_UNICODE[6028] := 16#90E4;
   // GBK_TO_UNICODE[6029] := 16#612A;
   // GBK_TO_UNICODE[6030] := 16#90E5;
   // GBK_TO_UNICODE[6031] := 16#612C;
   // GBK_TO_UNICODE[6032] := 16#90E6;
   // GBK_TO_UNICODE[6033] := 16#612D;
   // GBK_TO_UNICODE[6034] := 16#90E7;
   // GBK_TO_UNICODE[6035] := 16#612E;
   // GBK_TO_UNICODE[6036] := 16#90E8;
   // GBK_TO_UNICODE[6037] := 16#612F;
   // GBK_TO_UNICODE[6038] := 16#90E9;
   // GBK_TO_UNICODE[6039] := 16#6130;
   // GBK_TO_UNICODE[6040] := 16#90EA;
   // GBK_TO_UNICODE[6041] := 16#6131;
   // GBK_TO_UNICODE[6042] := 16#90EB;
   // GBK_TO_UNICODE[6043] := 16#6132;
   // GBK_TO_UNICODE[6044] := 16#90EC;
   // GBK_TO_UNICODE[6045] := 16#6133;
   // GBK_TO_UNICODE[6046] := 16#90ED;
   // GBK_TO_UNICODE[6047] := 16#6134;
   // GBK_TO_UNICODE[6048] := 16#90EE;
   // GBK_TO_UNICODE[6049] := 16#6135;
   // GBK_TO_UNICODE[6050] := 16#90EF;
   // GBK_TO_UNICODE[6051] := 16#6136;
   // GBK_TO_UNICODE[6052] := 16#90F0;
   // GBK_TO_UNICODE[6053] := 16#6137;
   // GBK_TO_UNICODE[6054] := 16#90F1;
   // GBK_TO_UNICODE[6055] := 16#6138;
   // GBK_TO_UNICODE[6056] := 16#90F2;
   // GBK_TO_UNICODE[6057] := 16#6139;
   // GBK_TO_UNICODE[6058] := 16#90F3;
   // GBK_TO_UNICODE[6059] := 16#613A;
   // GBK_TO_UNICODE[6060] := 16#90F4;
   // GBK_TO_UNICODE[6061] := 16#613B;
   // GBK_TO_UNICODE[6062] := 16#90F5;
   // GBK_TO_UNICODE[6063] := 16#613C;
   // GBK_TO_UNICODE[6064] := 16#90F6;
   // GBK_TO_UNICODE[6065] := 16#613D;
   // GBK_TO_UNICODE[6066] := 16#90F7;
   // GBK_TO_UNICODE[6067] := 16#613E;
   // GBK_TO_UNICODE[6068] := 16#90F8;
   // GBK_TO_UNICODE[6069] := 16#6140;
   // GBK_TO_UNICODE[6070] := 16#90F9;
   // GBK_TO_UNICODE[6071] := 16#6141;
   // GBK_TO_UNICODE[6072] := 16#90FA;
   // GBK_TO_UNICODE[6073] := 16#6142;
   // GBK_TO_UNICODE[6074] := 16#90FB;
   // GBK_TO_UNICODE[6075] := 16#6143;
   // GBK_TO_UNICODE[6076] := 16#90FC;
   // GBK_TO_UNICODE[6077] := 16#6144;
   // GBK_TO_UNICODE[6078] := 16#90FD;
   // GBK_TO_UNICODE[6079] := 16#6145;
   // GBK_TO_UNICODE[6080] := 16#90FE;
   // GBK_TO_UNICODE[6081] := 16#6146;
   // GBK_TO_UNICODE[6082] := 16#9140;
   // GBK_TO_UNICODE[6083] := 16#6147;
   // GBK_TO_UNICODE[6084] := 16#9141;
   // GBK_TO_UNICODE[6085] := 16#6149;
   // GBK_TO_UNICODE[6086] := 16#9142;
   // GBK_TO_UNICODE[6087] := 16#614B;
   // GBK_TO_UNICODE[6088] := 16#9143;
   // GBK_TO_UNICODE[6089] := 16#614D;
   // GBK_TO_UNICODE[6090] := 16#9144;
   // GBK_TO_UNICODE[6091] := 16#614F;
   // GBK_TO_UNICODE[6092] := 16#9145;
   // GBK_TO_UNICODE[6093] := 16#6150;
   // GBK_TO_UNICODE[6094] := 16#9146;
   // GBK_TO_UNICODE[6095] := 16#6152;
   // GBK_TO_UNICODE[6096] := 16#9147;
   // GBK_TO_UNICODE[6097] := 16#6153;
   // GBK_TO_UNICODE[6098] := 16#9148;
   // GBK_TO_UNICODE[6099] := 16#6154;
   // GBK_TO_UNICODE[6100] := 16#9149;
   // GBK_TO_UNICODE[6101] := 16#6156;
   // GBK_TO_UNICODE[6102] := 16#914A;
   // GBK_TO_UNICODE[6103] := 16#6157;
   // GBK_TO_UNICODE[6104] := 16#914B;
   // GBK_TO_UNICODE[6105] := 16#6158;
   // GBK_TO_UNICODE[6106] := 16#914C;
   // GBK_TO_UNICODE[6107] := 16#6159;
   // GBK_TO_UNICODE[6108] := 16#914D;
   // GBK_TO_UNICODE[6109] := 16#615A;
   // GBK_TO_UNICODE[6110] := 16#914E;
   // GBK_TO_UNICODE[6111] := 16#615B;
   // GBK_TO_UNICODE[6112] := 16#914F;
   // GBK_TO_UNICODE[6113] := 16#615C;
   // GBK_TO_UNICODE[6114] := 16#9150;
   // GBK_TO_UNICODE[6115] := 16#615E;
   // GBK_TO_UNICODE[6116] := 16#9151;
   // GBK_TO_UNICODE[6117] := 16#615F;
   // GBK_TO_UNICODE[6118] := 16#9152;
   // GBK_TO_UNICODE[6119] := 16#6160;
   // GBK_TO_UNICODE[6120] := 16#9153;
   // GBK_TO_UNICODE[6121] := 16#6161;
   // GBK_TO_UNICODE[6122] := 16#9154;
   // GBK_TO_UNICODE[6123] := 16#6163;
   // GBK_TO_UNICODE[6124] := 16#9155;
   // GBK_TO_UNICODE[6125] := 16#6164;
   // GBK_TO_UNICODE[6126] := 16#9156;
   // GBK_TO_UNICODE[6127] := 16#6165;
   // GBK_TO_UNICODE[6128] := 16#9157;
   // GBK_TO_UNICODE[6129] := 16#6166;
   // GBK_TO_UNICODE[6130] := 16#9158;
   // GBK_TO_UNICODE[6131] := 16#6169;
   // GBK_TO_UNICODE[6132] := 16#9159;
   // GBK_TO_UNICODE[6133] := 16#616A;
   // GBK_TO_UNICODE[6134] := 16#915A;
   // GBK_TO_UNICODE[6135] := 16#616B;
   // GBK_TO_UNICODE[6136] := 16#915B;
   // GBK_TO_UNICODE[6137] := 16#616C;
   // GBK_TO_UNICODE[6138] := 16#915C;
   // GBK_TO_UNICODE[6139] := 16#616D;
   // GBK_TO_UNICODE[6140] := 16#915D;
   // GBK_TO_UNICODE[6141] := 16#616E;
   // GBK_TO_UNICODE[6142] := 16#915E;
   // GBK_TO_UNICODE[6143] := 16#616F;
   // GBK_TO_UNICODE[6144] := 16#915F;
   // GBK_TO_UNICODE[6145] := 16#6171;
   // GBK_TO_UNICODE[6146] := 16#9160;
   // GBK_TO_UNICODE[6147] := 16#6172;
   // GBK_TO_UNICODE[6148] := 16#9161;
   // GBK_TO_UNICODE[6149] := 16#6173;
   // GBK_TO_UNICODE[6150] := 16#9162;
   // GBK_TO_UNICODE[6151] := 16#6174;
   // GBK_TO_UNICODE[6152] := 16#9163;
   // GBK_TO_UNICODE[6153] := 16#6176;
   // GBK_TO_UNICODE[6154] := 16#9164;
   // GBK_TO_UNICODE[6155] := 16#6178;
   // GBK_TO_UNICODE[6156] := 16#9165;
   // GBK_TO_UNICODE[6157] := 16#6179;
   // GBK_TO_UNICODE[6158] := 16#9166;
   // GBK_TO_UNICODE[6159] := 16#617A;
   // GBK_TO_UNICODE[6160] := 16#9167;
   // GBK_TO_UNICODE[6161] := 16#617B;
   // GBK_TO_UNICODE[6162] := 16#9168;
   // GBK_TO_UNICODE[6163] := 16#617C;
   // GBK_TO_UNICODE[6164] := 16#9169;
   // GBK_TO_UNICODE[6165] := 16#617D;
   // GBK_TO_UNICODE[6166] := 16#916A;
   // GBK_TO_UNICODE[6167] := 16#617E;
   // GBK_TO_UNICODE[6168] := 16#916B;
   // GBK_TO_UNICODE[6169] := 16#617F;
   // GBK_TO_UNICODE[6170] := 16#916C;
   // GBK_TO_UNICODE[6171] := 16#6180;
   // GBK_TO_UNICODE[6172] := 16#916D;
   // GBK_TO_UNICODE[6173] := 16#6181;
   // GBK_TO_UNICODE[6174] := 16#916E;
   // GBK_TO_UNICODE[6175] := 16#6182;
   // GBK_TO_UNICODE[6176] := 16#916F;
   // GBK_TO_UNICODE[6177] := 16#6183;
   // GBK_TO_UNICODE[6178] := 16#9170;
   // GBK_TO_UNICODE[6179] := 16#6184;
   // GBK_TO_UNICODE[6180] := 16#9171;
   // GBK_TO_UNICODE[6181] := 16#6185;
   // GBK_TO_UNICODE[6182] := 16#9172;
   // GBK_TO_UNICODE[6183] := 16#6186;
   // GBK_TO_UNICODE[6184] := 16#9173;
   // GBK_TO_UNICODE[6185] := 16#6187;
   // GBK_TO_UNICODE[6186] := 16#9174;
   // GBK_TO_UNICODE[6187] := 16#6188;
   // GBK_TO_UNICODE[6188] := 16#9175;
   // GBK_TO_UNICODE[6189] := 16#6189;
   // GBK_TO_UNICODE[6190] := 16#9176;
   // GBK_TO_UNICODE[6191] := 16#618A;
   // GBK_TO_UNICODE[6192] := 16#9177;
   // GBK_TO_UNICODE[6193] := 16#618C;
   // GBK_TO_UNICODE[6194] := 16#9178;
   // GBK_TO_UNICODE[6195] := 16#618D;
   // GBK_TO_UNICODE[6196] := 16#9179;
   // GBK_TO_UNICODE[6197] := 16#618F;
   // GBK_TO_UNICODE[6198] := 16#917A;
   // GBK_TO_UNICODE[6199] := 16#6190;
   // GBK_TO_UNICODE[6200] := 16#917B;
   // GBK_TO_UNICODE[6201] := 16#6191;
   // GBK_TO_UNICODE[6202] := 16#917C;
   // GBK_TO_UNICODE[6203] := 16#6192;
   // GBK_TO_UNICODE[6204] := 16#917D;
   // GBK_TO_UNICODE[6205] := 16#6193;
   // GBK_TO_UNICODE[6206] := 16#917E;
   // GBK_TO_UNICODE[6207] := 16#6195;
   // GBK_TO_UNICODE[6208] := 16#9180;
   // GBK_TO_UNICODE[6209] := 16#6196;
   // GBK_TO_UNICODE[6210] := 16#9181;
   // GBK_TO_UNICODE[6211] := 16#6197;
   // GBK_TO_UNICODE[6212] := 16#9182;
   // GBK_TO_UNICODE[6213] := 16#6198;
   // GBK_TO_UNICODE[6214] := 16#9183;
   // GBK_TO_UNICODE[6215] := 16#6199;
   // GBK_TO_UNICODE[6216] := 16#9184;
   // GBK_TO_UNICODE[6217] := 16#619A;
   // GBK_TO_UNICODE[6218] := 16#9185;
   // GBK_TO_UNICODE[6219] := 16#619B;
   // GBK_TO_UNICODE[6220] := 16#9186;
   // GBK_TO_UNICODE[6221] := 16#619C;
   // GBK_TO_UNICODE[6222] := 16#9187;
   // GBK_TO_UNICODE[6223] := 16#619E;
   // GBK_TO_UNICODE[6224] := 16#9188;
   // GBK_TO_UNICODE[6225] := 16#619F;
   // GBK_TO_UNICODE[6226] := 16#9189;
   // GBK_TO_UNICODE[6227] := 16#61A0;
   // GBK_TO_UNICODE[6228] := 16#918A;
   // GBK_TO_UNICODE[6229] := 16#61A1;
   // GBK_TO_UNICODE[6230] := 16#918B;
   // GBK_TO_UNICODE[6231] := 16#61A2;
   // GBK_TO_UNICODE[6232] := 16#918C;
   // GBK_TO_UNICODE[6233] := 16#61A3;
   // GBK_TO_UNICODE[6234] := 16#918D;
   // GBK_TO_UNICODE[6235] := 16#61A4;
   // GBK_TO_UNICODE[6236] := 16#918E;
   // GBK_TO_UNICODE[6237] := 16#61A5;
   // GBK_TO_UNICODE[6238] := 16#918F;
   // GBK_TO_UNICODE[6239] := 16#61A6;
   // GBK_TO_UNICODE[6240] := 16#9190;
   // GBK_TO_UNICODE[6241] := 16#61AA;
   // GBK_TO_UNICODE[6242] := 16#9191;
   // GBK_TO_UNICODE[6243] := 16#61AB;
   // GBK_TO_UNICODE[6244] := 16#9192;
   // GBK_TO_UNICODE[6245] := 16#61AD;
   // GBK_TO_UNICODE[6246] := 16#9193;
   // GBK_TO_UNICODE[6247] := 16#61AE;
   // GBK_TO_UNICODE[6248] := 16#9194;
   // GBK_TO_UNICODE[6249] := 16#61AF;
   // GBK_TO_UNICODE[6250] := 16#9195;
   // GBK_TO_UNICODE[6251] := 16#61B0;
   // GBK_TO_UNICODE[6252] := 16#9196;
   // GBK_TO_UNICODE[6253] := 16#61B1;
   // GBK_TO_UNICODE[6254] := 16#9197;
   // GBK_TO_UNICODE[6255] := 16#61B2;
   // GBK_TO_UNICODE[6256] := 16#9198;
   // GBK_TO_UNICODE[6257] := 16#61B3;
   // GBK_TO_UNICODE[6258] := 16#9199;
   // GBK_TO_UNICODE[6259] := 16#61B4;
   // GBK_TO_UNICODE[6260] := 16#919A;
   // GBK_TO_UNICODE[6261] := 16#61B5;
   // GBK_TO_UNICODE[6262] := 16#919B;
   // GBK_TO_UNICODE[6263] := 16#61B6;
   // GBK_TO_UNICODE[6264] := 16#919C;
   // GBK_TO_UNICODE[6265] := 16#61B8;
   // GBK_TO_UNICODE[6266] := 16#919D;
   // GBK_TO_UNICODE[6267] := 16#61B9;
   // GBK_TO_UNICODE[6268] := 16#919E;
   // GBK_TO_UNICODE[6269] := 16#61BA;
   // GBK_TO_UNICODE[6270] := 16#919F;
   // GBK_TO_UNICODE[6271] := 16#61BB;
   // GBK_TO_UNICODE[6272] := 16#91A0;
   // GBK_TO_UNICODE[6273] := 16#61BC;
   // GBK_TO_UNICODE[6274] := 16#91A1;
   // GBK_TO_UNICODE[6275] := 16#61BD;
   // GBK_TO_UNICODE[6276] := 16#91A2;
   // GBK_TO_UNICODE[6277] := 16#61BF;
   // GBK_TO_UNICODE[6278] := 16#91A3;
   // GBK_TO_UNICODE[6279] := 16#61C0;
   // GBK_TO_UNICODE[6280] := 16#91A4;
   // GBK_TO_UNICODE[6281] := 16#61C1;
   // GBK_TO_UNICODE[6282] := 16#91A5;
   // GBK_TO_UNICODE[6283] := 16#61C3;
   // GBK_TO_UNICODE[6284] := 16#91A6;
   // GBK_TO_UNICODE[6285] := 16#61C4;
   // GBK_TO_UNICODE[6286] := 16#91A7;
   // GBK_TO_UNICODE[6287] := 16#61C5;
   // GBK_TO_UNICODE[6288] := 16#91A8;
   // GBK_TO_UNICODE[6289] := 16#61C6;
   // GBK_TO_UNICODE[6290] := 16#91A9;
   // GBK_TO_UNICODE[6291] := 16#61C7;
   // GBK_TO_UNICODE[6292] := 16#91AA;
   // GBK_TO_UNICODE[6293] := 16#61C9;
   // GBK_TO_UNICODE[6294] := 16#91AB;
   // GBK_TO_UNICODE[6295] := 16#61CC;
   // GBK_TO_UNICODE[6296] := 16#91AC;
   // GBK_TO_UNICODE[6297] := 16#61CD;
   // GBK_TO_UNICODE[6298] := 16#91AD;
   // GBK_TO_UNICODE[6299] := 16#61CE;
   // GBK_TO_UNICODE[6300] := 16#91AE;
   // GBK_TO_UNICODE[6301] := 16#61CF;
   // GBK_TO_UNICODE[6302] := 16#91AF;
   // GBK_TO_UNICODE[6303] := 16#61D0;
   // GBK_TO_UNICODE[6304] := 16#91B0;
   // GBK_TO_UNICODE[6305] := 16#61D3;
   // GBK_TO_UNICODE[6306] := 16#91B1;
   // GBK_TO_UNICODE[6307] := 16#61D5;
   // GBK_TO_UNICODE[6308] := 16#91B2;
   // GBK_TO_UNICODE[6309] := 16#61D6;
   // GBK_TO_UNICODE[6310] := 16#91B3;
   // GBK_TO_UNICODE[6311] := 16#61D7;
   // GBK_TO_UNICODE[6312] := 16#91B4;
   // GBK_TO_UNICODE[6313] := 16#61D8;
   // GBK_TO_UNICODE[6314] := 16#91B5;
   // GBK_TO_UNICODE[6315] := 16#61D9;
   // GBK_TO_UNICODE[6316] := 16#91B6;
   // GBK_TO_UNICODE[6317] := 16#61DA;
   // GBK_TO_UNICODE[6318] := 16#91B7;
   // GBK_TO_UNICODE[6319] := 16#61DB;
   // GBK_TO_UNICODE[6320] := 16#91B8;
   // GBK_TO_UNICODE[6321] := 16#61DC;
   // GBK_TO_UNICODE[6322] := 16#91B9;
   // GBK_TO_UNICODE[6323] := 16#61DD;
   // GBK_TO_UNICODE[6324] := 16#91BA;
   // GBK_TO_UNICODE[6325] := 16#61DE;
   // GBK_TO_UNICODE[6326] := 16#91BB;
   // GBK_TO_UNICODE[6327] := 16#61DF;
   // GBK_TO_UNICODE[6328] := 16#91BC;
   // GBK_TO_UNICODE[6329] := 16#61E0;
   // GBK_TO_UNICODE[6330] := 16#91BD;
   // GBK_TO_UNICODE[6331] := 16#61E1;
   // GBK_TO_UNICODE[6332] := 16#91BE;
   // GBK_TO_UNICODE[6333] := 16#61E2;
   // GBK_TO_UNICODE[6334] := 16#91BF;
   // GBK_TO_UNICODE[6335] := 16#61E3;
   // GBK_TO_UNICODE[6336] := 16#91C0;
   // GBK_TO_UNICODE[6337] := 16#61E4;
   // GBK_TO_UNICODE[6338] := 16#91C1;
   // GBK_TO_UNICODE[6339] := 16#61E5;
   // GBK_TO_UNICODE[6340] := 16#91C2;
   // GBK_TO_UNICODE[6341] := 16#61E7;
   // GBK_TO_UNICODE[6342] := 16#91C3;
   // GBK_TO_UNICODE[6343] := 16#61E8;
   // GBK_TO_UNICODE[6344] := 16#91C4;
   // GBK_TO_UNICODE[6345] := 16#61E9;
   // GBK_TO_UNICODE[6346] := 16#91C5;
   // GBK_TO_UNICODE[6347] := 16#61EA;
   // GBK_TO_UNICODE[6348] := 16#91C6;
   // GBK_TO_UNICODE[6349] := 16#61EB;
   // GBK_TO_UNICODE[6350] := 16#91C7;
   // GBK_TO_UNICODE[6351] := 16#61EC;
   // GBK_TO_UNICODE[6352] := 16#91C8;
   // GBK_TO_UNICODE[6353] := 16#61ED;
   // GBK_TO_UNICODE[6354] := 16#91C9;
   // GBK_TO_UNICODE[6355] := 16#61EE;
   // GBK_TO_UNICODE[6356] := 16#91CA;
   // GBK_TO_UNICODE[6357] := 16#61EF;
   // GBK_TO_UNICODE[6358] := 16#91CB;
   // GBK_TO_UNICODE[6359] := 16#61F0;
   // GBK_TO_UNICODE[6360] := 16#91CC;
   // GBK_TO_UNICODE[6361] := 16#61F1;
   // GBK_TO_UNICODE[6362] := 16#91CD;
   // GBK_TO_UNICODE[6363] := 16#61F2;
   // GBK_TO_UNICODE[6364] := 16#91CE;
   // GBK_TO_UNICODE[6365] := 16#61F3;
   // GBK_TO_UNICODE[6366] := 16#91CF;
   // GBK_TO_UNICODE[6367] := 16#61F4;
   // GBK_TO_UNICODE[6368] := 16#91D0;
   // GBK_TO_UNICODE[6369] := 16#61F6;
   // GBK_TO_UNICODE[6370] := 16#91D1;
   // GBK_TO_UNICODE[6371] := 16#61F7;
   // GBK_TO_UNICODE[6372] := 16#91D2;
   // GBK_TO_UNICODE[6373] := 16#61F8;
   // GBK_TO_UNICODE[6374] := 16#91D3;
   // GBK_TO_UNICODE[6375] := 16#61F9;
   // GBK_TO_UNICODE[6376] := 16#91D4;
   // GBK_TO_UNICODE[6377] := 16#61FA;
   // GBK_TO_UNICODE[6378] := 16#91D5;
   // GBK_TO_UNICODE[6379] := 16#61FB;
   // GBK_TO_UNICODE[6380] := 16#91D6;
   // GBK_TO_UNICODE[6381] := 16#61FC;
   // GBK_TO_UNICODE[6382] := 16#91D7;
   // GBK_TO_UNICODE[6383] := 16#61FD;
   // GBK_TO_UNICODE[6384] := 16#91D8;
   // GBK_TO_UNICODE[6385] := 16#61FE;
   // GBK_TO_UNICODE[6386] := 16#91D9;
   // GBK_TO_UNICODE[6387] := 16#6200;
   // GBK_TO_UNICODE[6388] := 16#91DA;
   // GBK_TO_UNICODE[6389] := 16#6201;
   // GBK_TO_UNICODE[6390] := 16#91DB;
   // GBK_TO_UNICODE[6391] := 16#6202;
   // GBK_TO_UNICODE[6392] := 16#91DC;
   // GBK_TO_UNICODE[6393] := 16#6203;
   // GBK_TO_UNICODE[6394] := 16#91DD;
   // GBK_TO_UNICODE[6395] := 16#6204;
   // GBK_TO_UNICODE[6396] := 16#91DE;
   // GBK_TO_UNICODE[6397] := 16#6205;
   // GBK_TO_UNICODE[6398] := 16#91DF;
   // GBK_TO_UNICODE[6399] := 16#6207;
   // GBK_TO_UNICODE[6400] := 16#91E0;
   // GBK_TO_UNICODE[6401] := 16#6209;
   // GBK_TO_UNICODE[6402] := 16#91E1;
   // GBK_TO_UNICODE[6403] := 16#6213;
   // GBK_TO_UNICODE[6404] := 16#91E2;
   // GBK_TO_UNICODE[6405] := 16#6214;
   // GBK_TO_UNICODE[6406] := 16#91E3;
   // GBK_TO_UNICODE[6407] := 16#6219;
   // GBK_TO_UNICODE[6408] := 16#91E4;
   // GBK_TO_UNICODE[6409] := 16#621C;
   // GBK_TO_UNICODE[6410] := 16#91E5;
   // GBK_TO_UNICODE[6411] := 16#621D;
   // GBK_TO_UNICODE[6412] := 16#91E6;
   // GBK_TO_UNICODE[6413] := 16#621E;
   // GBK_TO_UNICODE[6414] := 16#91E7;
   // GBK_TO_UNICODE[6415] := 16#6220;
   // GBK_TO_UNICODE[6416] := 16#91E8;
   // GBK_TO_UNICODE[6417] := 16#6223;
   // GBK_TO_UNICODE[6418] := 16#91E9;
   // GBK_TO_UNICODE[6419] := 16#6226;
   // GBK_TO_UNICODE[6420] := 16#91EA;
   // GBK_TO_UNICODE[6421] := 16#6227;
   // GBK_TO_UNICODE[6422] := 16#91EB;
   // GBK_TO_UNICODE[6423] := 16#6228;
   // GBK_TO_UNICODE[6424] := 16#91EC;
   // GBK_TO_UNICODE[6425] := 16#6229;
   // GBK_TO_UNICODE[6426] := 16#91ED;
   // GBK_TO_UNICODE[6427] := 16#622B;
   // GBK_TO_UNICODE[6428] := 16#91EE;
   // GBK_TO_UNICODE[6429] := 16#622D;
   // GBK_TO_UNICODE[6430] := 16#91EF;
   // GBK_TO_UNICODE[6431] := 16#622F;
   // GBK_TO_UNICODE[6432] := 16#91F0;
   // GBK_TO_UNICODE[6433] := 16#6230;
   // GBK_TO_UNICODE[6434] := 16#91F1;
   // GBK_TO_UNICODE[6435] := 16#6231;
   // GBK_TO_UNICODE[6436] := 16#91F2;
   // GBK_TO_UNICODE[6437] := 16#6232;
   // GBK_TO_UNICODE[6438] := 16#91F3;
   // GBK_TO_UNICODE[6439] := 16#6235;
   // GBK_TO_UNICODE[6440] := 16#91F4;
   // GBK_TO_UNICODE[6441] := 16#6236;
   // GBK_TO_UNICODE[6442] := 16#91F5;
   // GBK_TO_UNICODE[6443] := 16#6238;
   // GBK_TO_UNICODE[6444] := 16#91F6;
   // GBK_TO_UNICODE[6445] := 16#6239;
   // GBK_TO_UNICODE[6446] := 16#91F7;
   // GBK_TO_UNICODE[6447] := 16#623A;
   // GBK_TO_UNICODE[6448] := 16#91F8;
   // GBK_TO_UNICODE[6449] := 16#623B;
   // GBK_TO_UNICODE[6450] := 16#91F9;
   // GBK_TO_UNICODE[6451] := 16#623C;
   // GBK_TO_UNICODE[6452] := 16#91FA;
   // GBK_TO_UNICODE[6453] := 16#6242;
   // GBK_TO_UNICODE[6454] := 16#91FB;
   // GBK_TO_UNICODE[6455] := 16#6244;
   // GBK_TO_UNICODE[6456] := 16#91FC;
   // GBK_TO_UNICODE[6457] := 16#6245;
   // GBK_TO_UNICODE[6458] := 16#91FD;
   // GBK_TO_UNICODE[6459] := 16#6246;
   // GBK_TO_UNICODE[6460] := 16#91FE;
   // GBK_TO_UNICODE[6461] := 16#624A;
   // GBK_TO_UNICODE[6462] := 16#9240;
   // GBK_TO_UNICODE[6463] := 16#624F;
   // GBK_TO_UNICODE[6464] := 16#9241;
   // GBK_TO_UNICODE[6465] := 16#6250;
   // GBK_TO_UNICODE[6466] := 16#9242;
   // GBK_TO_UNICODE[6467] := 16#6255;
   // GBK_TO_UNICODE[6468] := 16#9243;
   // GBK_TO_UNICODE[6469] := 16#6256;
   // GBK_TO_UNICODE[6470] := 16#9244;
   // GBK_TO_UNICODE[6471] := 16#6257;
   // GBK_TO_UNICODE[6472] := 16#9245;
   // GBK_TO_UNICODE[6473] := 16#6259;
   // GBK_TO_UNICODE[6474] := 16#9246;
   // GBK_TO_UNICODE[6475] := 16#625A;
   // GBK_TO_UNICODE[6476] := 16#9247;
   // GBK_TO_UNICODE[6477] := 16#625C;
   // GBK_TO_UNICODE[6478] := 16#9248;
   // GBK_TO_UNICODE[6479] := 16#625D;
   // GBK_TO_UNICODE[6480] := 16#9249;
   // GBK_TO_UNICODE[6481] := 16#625E;
   // GBK_TO_UNICODE[6482] := 16#924A;
   // GBK_TO_UNICODE[6483] := 16#625F;
   // GBK_TO_UNICODE[6484] := 16#924B;
   // GBK_TO_UNICODE[6485] := 16#6260;
   // GBK_TO_UNICODE[6486] := 16#924C;
   // GBK_TO_UNICODE[6487] := 16#6261;
   // GBK_TO_UNICODE[6488] := 16#924D;
   // GBK_TO_UNICODE[6489] := 16#6262;
   // GBK_TO_UNICODE[6490] := 16#924E;
   // GBK_TO_UNICODE[6491] := 16#6264;
   // GBK_TO_UNICODE[6492] := 16#924F;
   // GBK_TO_UNICODE[6493] := 16#6265;
   // GBK_TO_UNICODE[6494] := 16#9250;
   // GBK_TO_UNICODE[6495] := 16#6268;
   // GBK_TO_UNICODE[6496] := 16#9251;
   // GBK_TO_UNICODE[6497] := 16#6271;
   // GBK_TO_UNICODE[6498] := 16#9252;
   // GBK_TO_UNICODE[6499] := 16#6272;
   // GBK_TO_UNICODE[6500] := 16#9253;
   // GBK_TO_UNICODE[6501] := 16#6274;
   // GBK_TO_UNICODE[6502] := 16#9254;
   // GBK_TO_UNICODE[6503] := 16#6275;
   // GBK_TO_UNICODE[6504] := 16#9255;
   // GBK_TO_UNICODE[6505] := 16#6277;
   // GBK_TO_UNICODE[6506] := 16#9256;
   // GBK_TO_UNICODE[6507] := 16#6278;
   // GBK_TO_UNICODE[6508] := 16#9257;
   // GBK_TO_UNICODE[6509] := 16#627A;
   // GBK_TO_UNICODE[6510] := 16#9258;
   // GBK_TO_UNICODE[6511] := 16#627B;
   // GBK_TO_UNICODE[6512] := 16#9259;
   // GBK_TO_UNICODE[6513] := 16#627D;
   // GBK_TO_UNICODE[6514] := 16#925A;
   // GBK_TO_UNICODE[6515] := 16#6281;
   // GBK_TO_UNICODE[6516] := 16#925B;
   // GBK_TO_UNICODE[6517] := 16#6282;
   // GBK_TO_UNICODE[6518] := 16#925C;
   // GBK_TO_UNICODE[6519] := 16#6283;
   // GBK_TO_UNICODE[6520] := 16#925D;
   // GBK_TO_UNICODE[6521] := 16#6285;
   // GBK_TO_UNICODE[6522] := 16#925E;
   // GBK_TO_UNICODE[6523] := 16#6286;
   // GBK_TO_UNICODE[6524] := 16#925F;
   // GBK_TO_UNICODE[6525] := 16#6287;
   // GBK_TO_UNICODE[6526] := 16#9260;
   // GBK_TO_UNICODE[6527] := 16#6288;
   // GBK_TO_UNICODE[6528] := 16#9261;
   // GBK_TO_UNICODE[6529] := 16#628B;
   // GBK_TO_UNICODE[6530] := 16#9262;
   // GBK_TO_UNICODE[6531] := 16#628C;
   // GBK_TO_UNICODE[6532] := 16#9263;
   // GBK_TO_UNICODE[6533] := 16#628D;
   // GBK_TO_UNICODE[6534] := 16#9264;
   // GBK_TO_UNICODE[6535] := 16#628E;
   // GBK_TO_UNICODE[6536] := 16#9265;
   // GBK_TO_UNICODE[6537] := 16#628F;
   // GBK_TO_UNICODE[6538] := 16#9266;
   // GBK_TO_UNICODE[6539] := 16#6290;
   // GBK_TO_UNICODE[6540] := 16#9267;
   // GBK_TO_UNICODE[6541] := 16#6294;
   // GBK_TO_UNICODE[6542] := 16#9268;
   // GBK_TO_UNICODE[6543] := 16#6299;
   // GBK_TO_UNICODE[6544] := 16#9269;
   // GBK_TO_UNICODE[6545] := 16#629C;
   // GBK_TO_UNICODE[6546] := 16#926A;
   // GBK_TO_UNICODE[6547] := 16#629D;
   // GBK_TO_UNICODE[6548] := 16#926B;
   // GBK_TO_UNICODE[6549] := 16#629E;
   // GBK_TO_UNICODE[6550] := 16#926C;
   // GBK_TO_UNICODE[6551] := 16#62A3;
   // GBK_TO_UNICODE[6552] := 16#926D;
   // GBK_TO_UNICODE[6553] := 16#62A6;
   // GBK_TO_UNICODE[6554] := 16#926E;
   // GBK_TO_UNICODE[6555] := 16#62A7;
   // GBK_TO_UNICODE[6556] := 16#926F;
   // GBK_TO_UNICODE[6557] := 16#62A9;
   // GBK_TO_UNICODE[6558] := 16#9270;
   // GBK_TO_UNICODE[6559] := 16#62AA;
   // GBK_TO_UNICODE[6560] := 16#9271;
   // GBK_TO_UNICODE[6561] := 16#62AD;
   // GBK_TO_UNICODE[6562] := 16#9272;
   // GBK_TO_UNICODE[6563] := 16#62AE;
   // GBK_TO_UNICODE[6564] := 16#9273;
   // GBK_TO_UNICODE[6565] := 16#62AF;
   // GBK_TO_UNICODE[6566] := 16#9274;
   // GBK_TO_UNICODE[6567] := 16#62B0;
   // GBK_TO_UNICODE[6568] := 16#9275;
   // GBK_TO_UNICODE[6569] := 16#62B2;
   // GBK_TO_UNICODE[6570] := 16#9276;
   // GBK_TO_UNICODE[6571] := 16#62B3;
   // GBK_TO_UNICODE[6572] := 16#9277;
   // GBK_TO_UNICODE[6573] := 16#62B4;
   // GBK_TO_UNICODE[6574] := 16#9278;
   // GBK_TO_UNICODE[6575] := 16#62B6;
   // GBK_TO_UNICODE[6576] := 16#9279;
   // GBK_TO_UNICODE[6577] := 16#62B7;
   // GBK_TO_UNICODE[6578] := 16#927A;
   // GBK_TO_UNICODE[6579] := 16#62B8;
   // GBK_TO_UNICODE[6580] := 16#927B;
   // GBK_TO_UNICODE[6581] := 16#62BA;
   // GBK_TO_UNICODE[6582] := 16#927C;
   // GBK_TO_UNICODE[6583] := 16#62BE;
   // GBK_TO_UNICODE[6584] := 16#927D;
   // GBK_TO_UNICODE[6585] := 16#62C0;
   // GBK_TO_UNICODE[6586] := 16#927E;
   // GBK_TO_UNICODE[6587] := 16#62C1;
   // GBK_TO_UNICODE[6588] := 16#9280;
   // GBK_TO_UNICODE[6589] := 16#62C3;
   // GBK_TO_UNICODE[6590] := 16#9281;
   // GBK_TO_UNICODE[6591] := 16#62CB;
   // GBK_TO_UNICODE[6592] := 16#9282;
   // GBK_TO_UNICODE[6593] := 16#62CF;
   // GBK_TO_UNICODE[6594] := 16#9283;
   // GBK_TO_UNICODE[6595] := 16#62D1;
   // GBK_TO_UNICODE[6596] := 16#9284;
   // GBK_TO_UNICODE[6597] := 16#62D5;
   // GBK_TO_UNICODE[6598] := 16#9285;
   // GBK_TO_UNICODE[6599] := 16#62DD;
   // GBK_TO_UNICODE[6600] := 16#9286;
   // GBK_TO_UNICODE[6601] := 16#62DE;
   // GBK_TO_UNICODE[6602] := 16#9287;
   // GBK_TO_UNICODE[6603] := 16#62E0;
   // GBK_TO_UNICODE[6604] := 16#9288;
   // GBK_TO_UNICODE[6605] := 16#62E1;
   // GBK_TO_UNICODE[6606] := 16#9289;
   // GBK_TO_UNICODE[6607] := 16#62E4;
   // GBK_TO_UNICODE[6608] := 16#928A;
   // GBK_TO_UNICODE[6609] := 16#62EA;
   // GBK_TO_UNICODE[6610] := 16#928B;
   // GBK_TO_UNICODE[6611] := 16#62EB;
   // GBK_TO_UNICODE[6612] := 16#928C;
   // GBK_TO_UNICODE[6613] := 16#62F0;
   // GBK_TO_UNICODE[6614] := 16#928D;
   // GBK_TO_UNICODE[6615] := 16#62F2;
   // GBK_TO_UNICODE[6616] := 16#928E;
   // GBK_TO_UNICODE[6617] := 16#62F5;
   // GBK_TO_UNICODE[6618] := 16#928F;
   // GBK_TO_UNICODE[6619] := 16#62F8;
   // GBK_TO_UNICODE[6620] := 16#9290;
   // GBK_TO_UNICODE[6621] := 16#62F9;
   // GBK_TO_UNICODE[6622] := 16#9291;
   // GBK_TO_UNICODE[6623] := 16#62FA;
   // GBK_TO_UNICODE[6624] := 16#9292;
   // GBK_TO_UNICODE[6625] := 16#62FB;
   // GBK_TO_UNICODE[6626] := 16#9293;
   // GBK_TO_UNICODE[6627] := 16#6300;
   // GBK_TO_UNICODE[6628] := 16#9294;
   // GBK_TO_UNICODE[6629] := 16#6303;
   // GBK_TO_UNICODE[6630] := 16#9295;
   // GBK_TO_UNICODE[6631] := 16#6304;
   // GBK_TO_UNICODE[6632] := 16#9296;
   // GBK_TO_UNICODE[6633] := 16#6305;
   // GBK_TO_UNICODE[6634] := 16#9297;
   // GBK_TO_UNICODE[6635] := 16#6306;
   // GBK_TO_UNICODE[6636] := 16#9298;
   // GBK_TO_UNICODE[6637] := 16#630A;
   // GBK_TO_UNICODE[6638] := 16#9299;
   // GBK_TO_UNICODE[6639] := 16#630B;
   // GBK_TO_UNICODE[6640] := 16#929A;
   // GBK_TO_UNICODE[6641] := 16#630C;
   // GBK_TO_UNICODE[6642] := 16#929B;
   // GBK_TO_UNICODE[6643] := 16#630D;
   // GBK_TO_UNICODE[6644] := 16#929C;
   // GBK_TO_UNICODE[6645] := 16#630F;
   // GBK_TO_UNICODE[6646] := 16#929D;
   // GBK_TO_UNICODE[6647] := 16#6310;
   // GBK_TO_UNICODE[6648] := 16#929E;
   // GBK_TO_UNICODE[6649] := 16#6312;
   // GBK_TO_UNICODE[6650] := 16#929F;
   // GBK_TO_UNICODE[6651] := 16#6313;
   // GBK_TO_UNICODE[6652] := 16#92A0;
   // GBK_TO_UNICODE[6653] := 16#6314;
   // GBK_TO_UNICODE[6654] := 16#92A1;
   // GBK_TO_UNICODE[6655] := 16#6315;
   // GBK_TO_UNICODE[6656] := 16#92A2;
   // GBK_TO_UNICODE[6657] := 16#6317;
   // GBK_TO_UNICODE[6658] := 16#92A3;
   // GBK_TO_UNICODE[6659] := 16#6318;
   // GBK_TO_UNICODE[6660] := 16#92A4;
   // GBK_TO_UNICODE[6661] := 16#6319;
   // GBK_TO_UNICODE[6662] := 16#92A5;
   // GBK_TO_UNICODE[6663] := 16#631C;
   // GBK_TO_UNICODE[6664] := 16#92A6;
   // GBK_TO_UNICODE[6665] := 16#6326;
   // GBK_TO_UNICODE[6666] := 16#92A7;
   // GBK_TO_UNICODE[6667] := 16#6327;
   // GBK_TO_UNICODE[6668] := 16#92A8;
   // GBK_TO_UNICODE[6669] := 16#6329;
   // GBK_TO_UNICODE[6670] := 16#92A9;
   // GBK_TO_UNICODE[6671] := 16#632C;
   // GBK_TO_UNICODE[6672] := 16#92AA;
   // GBK_TO_UNICODE[6673] := 16#632D;
   // GBK_TO_UNICODE[6674] := 16#92AB;
   // GBK_TO_UNICODE[6675] := 16#632E;
   // GBK_TO_UNICODE[6676] := 16#92AC;
   // GBK_TO_UNICODE[6677] := 16#6330;
   // GBK_TO_UNICODE[6678] := 16#92AD;
   // GBK_TO_UNICODE[6679] := 16#6331;
   // GBK_TO_UNICODE[6680] := 16#92AE;
   // GBK_TO_UNICODE[6681] := 16#6333;
   // GBK_TO_UNICODE[6682] := 16#92AF;
   // GBK_TO_UNICODE[6683] := 16#6334;
   // GBK_TO_UNICODE[6684] := 16#92B0;
   // GBK_TO_UNICODE[6685] := 16#6335;
   // GBK_TO_UNICODE[6686] := 16#92B1;
   // GBK_TO_UNICODE[6687] := 16#6336;
   // GBK_TO_UNICODE[6688] := 16#92B2;
   // GBK_TO_UNICODE[6689] := 16#6337;
   // GBK_TO_UNICODE[6690] := 16#92B3;
   // GBK_TO_UNICODE[6691] := 16#6338;
   // GBK_TO_UNICODE[6692] := 16#92B4;
   // GBK_TO_UNICODE[6693] := 16#633B;
   // GBK_TO_UNICODE[6694] := 16#92B5;
   // GBK_TO_UNICODE[6695] := 16#633C;
   // GBK_TO_UNICODE[6696] := 16#92B6;
   // GBK_TO_UNICODE[6697] := 16#633E;
   // GBK_TO_UNICODE[6698] := 16#92B7;
   // GBK_TO_UNICODE[6699] := 16#633F;
   // GBK_TO_UNICODE[6700] := 16#92B8;
   // GBK_TO_UNICODE[6701] := 16#6340;
   // GBK_TO_UNICODE[6702] := 16#92B9;
   // GBK_TO_UNICODE[6703] := 16#6341;
   // GBK_TO_UNICODE[6704] := 16#92BA;
   // GBK_TO_UNICODE[6705] := 16#6344;
   // GBK_TO_UNICODE[6706] := 16#92BB;
   // GBK_TO_UNICODE[6707] := 16#6347;
   // GBK_TO_UNICODE[6708] := 16#92BC;
   // GBK_TO_UNICODE[6709] := 16#6348;
   // GBK_TO_UNICODE[6710] := 16#92BD;
   // GBK_TO_UNICODE[6711] := 16#634A;
   // GBK_TO_UNICODE[6712] := 16#92BE;
   // GBK_TO_UNICODE[6713] := 16#6351;
   // GBK_TO_UNICODE[6714] := 16#92BF;
   // GBK_TO_UNICODE[6715] := 16#6352;
   // GBK_TO_UNICODE[6716] := 16#92C0;
   // GBK_TO_UNICODE[6717] := 16#6353;
   // GBK_TO_UNICODE[6718] := 16#92C1;
   // GBK_TO_UNICODE[6719] := 16#6354;
   // GBK_TO_UNICODE[6720] := 16#92C2;
   // GBK_TO_UNICODE[6721] := 16#6356;
   // GBK_TO_UNICODE[6722] := 16#92C3;
   // GBK_TO_UNICODE[6723] := 16#6357;
   // GBK_TO_UNICODE[6724] := 16#92C4;
   // GBK_TO_UNICODE[6725] := 16#6358;
   // GBK_TO_UNICODE[6726] := 16#92C5;
   // GBK_TO_UNICODE[6727] := 16#6359;
   // GBK_TO_UNICODE[6728] := 16#92C6;
   // GBK_TO_UNICODE[6729] := 16#635A;
   // GBK_TO_UNICODE[6730] := 16#92C7;
   // GBK_TO_UNICODE[6731] := 16#635B;
   // GBK_TO_UNICODE[6732] := 16#92C8;
   // GBK_TO_UNICODE[6733] := 16#635C;
   // GBK_TO_UNICODE[6734] := 16#92C9;
   // GBK_TO_UNICODE[6735] := 16#635D;
   // GBK_TO_UNICODE[6736] := 16#92CA;
   // GBK_TO_UNICODE[6737] := 16#6360;
   // GBK_TO_UNICODE[6738] := 16#92CB;
   // GBK_TO_UNICODE[6739] := 16#6364;
   // GBK_TO_UNICODE[6740] := 16#92CC;
   // GBK_TO_UNICODE[6741] := 16#6365;
   // GBK_TO_UNICODE[6742] := 16#92CD;
   // GBK_TO_UNICODE[6743] := 16#6366;
   // GBK_TO_UNICODE[6744] := 16#92CE;
   // GBK_TO_UNICODE[6745] := 16#6368;
   // GBK_TO_UNICODE[6746] := 16#92CF;
   // GBK_TO_UNICODE[6747] := 16#636A;
   // GBK_TO_UNICODE[6748] := 16#92D0;
   // GBK_TO_UNICODE[6749] := 16#636B;
   // GBK_TO_UNICODE[6750] := 16#92D1;
   // GBK_TO_UNICODE[6751] := 16#636C;
   // GBK_TO_UNICODE[6752] := 16#92D2;
   // GBK_TO_UNICODE[6753] := 16#636F;
   // GBK_TO_UNICODE[6754] := 16#92D3;
   // GBK_TO_UNICODE[6755] := 16#6370;
   // GBK_TO_UNICODE[6756] := 16#92D4;
   // GBK_TO_UNICODE[6757] := 16#6372;
   // GBK_TO_UNICODE[6758] := 16#92D5;
   // GBK_TO_UNICODE[6759] := 16#6373;
   // GBK_TO_UNICODE[6760] := 16#92D6;
   // GBK_TO_UNICODE[6761] := 16#6374;
   // GBK_TO_UNICODE[6762] := 16#92D7;
   // GBK_TO_UNICODE[6763] := 16#6375;
   // GBK_TO_UNICODE[6764] := 16#92D8;
   // GBK_TO_UNICODE[6765] := 16#6378;
   // GBK_TO_UNICODE[6766] := 16#92D9;
   // GBK_TO_UNICODE[6767] := 16#6379;
   // GBK_TO_UNICODE[6768] := 16#92DA;
   // GBK_TO_UNICODE[6769] := 16#637C;
   // GBK_TO_UNICODE[6770] := 16#92DB;
   // GBK_TO_UNICODE[6771] := 16#637D;
   // GBK_TO_UNICODE[6772] := 16#92DC;
   // GBK_TO_UNICODE[6773] := 16#637E;
   // GBK_TO_UNICODE[6774] := 16#92DD;
   // GBK_TO_UNICODE[6775] := 16#637F;
   // GBK_TO_UNICODE[6776] := 16#92DE;
   // GBK_TO_UNICODE[6777] := 16#6381;
   // GBK_TO_UNICODE[6778] := 16#92DF;
   // GBK_TO_UNICODE[6779] := 16#6383;
   // GBK_TO_UNICODE[6780] := 16#92E0;
   // GBK_TO_UNICODE[6781] := 16#6384;
   // GBK_TO_UNICODE[6782] := 16#92E1;
   // GBK_TO_UNICODE[6783] := 16#6385;
   // GBK_TO_UNICODE[6784] := 16#92E2;
   // GBK_TO_UNICODE[6785] := 16#6386;
   // GBK_TO_UNICODE[6786] := 16#92E3;
   // GBK_TO_UNICODE[6787] := 16#638B;
   // GBK_TO_UNICODE[6788] := 16#92E4;
   // GBK_TO_UNICODE[6789] := 16#638D;
   // GBK_TO_UNICODE[6790] := 16#92E5;
   // GBK_TO_UNICODE[6791] := 16#6391;
   // GBK_TO_UNICODE[6792] := 16#92E6;
   // GBK_TO_UNICODE[6793] := 16#6393;
   // GBK_TO_UNICODE[6794] := 16#92E7;
   // GBK_TO_UNICODE[6795] := 16#6394;
   // GBK_TO_UNICODE[6796] := 16#92E8;
   // GBK_TO_UNICODE[6797] := 16#6395;
   // GBK_TO_UNICODE[6798] := 16#92E9;
   // GBK_TO_UNICODE[6799] := 16#6397;
   // GBK_TO_UNICODE[6800] := 16#92EA;
   // GBK_TO_UNICODE[6801] := 16#6399;
   // GBK_TO_UNICODE[6802] := 16#92EB;
   // GBK_TO_UNICODE[6803] := 16#639A;
   // GBK_TO_UNICODE[6804] := 16#92EC;
   // GBK_TO_UNICODE[6805] := 16#639B;
   // GBK_TO_UNICODE[6806] := 16#92ED;
   // GBK_TO_UNICODE[6807] := 16#639C;
   // GBK_TO_UNICODE[6808] := 16#92EE;
   // GBK_TO_UNICODE[6809] := 16#639D;
   // GBK_TO_UNICODE[6810] := 16#92EF;
   // GBK_TO_UNICODE[6811] := 16#639E;
   // GBK_TO_UNICODE[6812] := 16#92F0;
   // GBK_TO_UNICODE[6813] := 16#639F;
   // GBK_TO_UNICODE[6814] := 16#92F1;
   // GBK_TO_UNICODE[6815] := 16#63A1;
   // GBK_TO_UNICODE[6816] := 16#92F2;
   // GBK_TO_UNICODE[6817] := 16#63A4;
   // GBK_TO_UNICODE[6818] := 16#92F3;
   // GBK_TO_UNICODE[6819] := 16#63A6;
   // GBK_TO_UNICODE[6820] := 16#92F4;
   // GBK_TO_UNICODE[6821] := 16#63AB;
   // GBK_TO_UNICODE[6822] := 16#92F5;
   // GBK_TO_UNICODE[6823] := 16#63AF;
   // GBK_TO_UNICODE[6824] := 16#92F6;
   // GBK_TO_UNICODE[6825] := 16#63B1;
   // GBK_TO_UNICODE[6826] := 16#92F7;
   // GBK_TO_UNICODE[6827] := 16#63B2;
   // GBK_TO_UNICODE[6828] := 16#92F8;
   // GBK_TO_UNICODE[6829] := 16#63B5;
   // GBK_TO_UNICODE[6830] := 16#92F9;
   // GBK_TO_UNICODE[6831] := 16#63B6;
   // GBK_TO_UNICODE[6832] := 16#92FA;
   // GBK_TO_UNICODE[6833] := 16#63B9;
   // GBK_TO_UNICODE[6834] := 16#92FB;
   // GBK_TO_UNICODE[6835] := 16#63BB;
   // GBK_TO_UNICODE[6836] := 16#92FC;
   // GBK_TO_UNICODE[6837] := 16#63BD;
   // GBK_TO_UNICODE[6838] := 16#92FD;
   // GBK_TO_UNICODE[6839] := 16#63BF;
   // GBK_TO_UNICODE[6840] := 16#92FE;
   // GBK_TO_UNICODE[6841] := 16#63C0;
   // GBK_TO_UNICODE[6842] := 16#9340;
   // GBK_TO_UNICODE[6843] := 16#63C1;
   // GBK_TO_UNICODE[6844] := 16#9341;
   // GBK_TO_UNICODE[6845] := 16#63C2;
   // GBK_TO_UNICODE[6846] := 16#9342;
   // GBK_TO_UNICODE[6847] := 16#63C3;
   // GBK_TO_UNICODE[6848] := 16#9343;
   // GBK_TO_UNICODE[6849] := 16#63C5;
   // GBK_TO_UNICODE[6850] := 16#9344;
   // GBK_TO_UNICODE[6851] := 16#63C7;
   // GBK_TO_UNICODE[6852] := 16#9345;
   // GBK_TO_UNICODE[6853] := 16#63C8;
   // GBK_TO_UNICODE[6854] := 16#9346;
   // GBK_TO_UNICODE[6855] := 16#63CA;
   // GBK_TO_UNICODE[6856] := 16#9347;
   // GBK_TO_UNICODE[6857] := 16#63CB;
   // GBK_TO_UNICODE[6858] := 16#9348;
   // GBK_TO_UNICODE[6859] := 16#63CC;
   // GBK_TO_UNICODE[6860] := 16#9349;
   // GBK_TO_UNICODE[6861] := 16#63D1;
   // GBK_TO_UNICODE[6862] := 16#934A;
   // GBK_TO_UNICODE[6863] := 16#63D3;
   // GBK_TO_UNICODE[6864] := 16#934B;
   // GBK_TO_UNICODE[6865] := 16#63D4;
   // GBK_TO_UNICODE[6866] := 16#934C;
   // GBK_TO_UNICODE[6867] := 16#63D5;
   // GBK_TO_UNICODE[6868] := 16#934D;
   // GBK_TO_UNICODE[6869] := 16#63D7;
   // GBK_TO_UNICODE[6870] := 16#934E;
   // GBK_TO_UNICODE[6871] := 16#63D8;
   // GBK_TO_UNICODE[6872] := 16#934F;
   // GBK_TO_UNICODE[6873] := 16#63D9;
   // GBK_TO_UNICODE[6874] := 16#9350;
   // GBK_TO_UNICODE[6875] := 16#63DA;
   // GBK_TO_UNICODE[6876] := 16#9351;
   // GBK_TO_UNICODE[6877] := 16#63DB;
   // GBK_TO_UNICODE[6878] := 16#9352;
   // GBK_TO_UNICODE[6879] := 16#63DC;
   // GBK_TO_UNICODE[6880] := 16#9353;
   // GBK_TO_UNICODE[6881] := 16#63DD;
   // GBK_TO_UNICODE[6882] := 16#9354;
   // GBK_TO_UNICODE[6883] := 16#63DF;
   // GBK_TO_UNICODE[6884] := 16#9355;
   // GBK_TO_UNICODE[6885] := 16#63E2;
   // GBK_TO_UNICODE[6886] := 16#9356;
   // GBK_TO_UNICODE[6887] := 16#63E4;
   // GBK_TO_UNICODE[6888] := 16#9357;
   // GBK_TO_UNICODE[6889] := 16#63E5;
   // GBK_TO_UNICODE[6890] := 16#9358;
   // GBK_TO_UNICODE[6891] := 16#63E6;
   // GBK_TO_UNICODE[6892] := 16#9359;
   // GBK_TO_UNICODE[6893] := 16#63E7;
   // GBK_TO_UNICODE[6894] := 16#935A;
   // GBK_TO_UNICODE[6895] := 16#63E8;
   // GBK_TO_UNICODE[6896] := 16#935B;
   // GBK_TO_UNICODE[6897] := 16#63EB;
   // GBK_TO_UNICODE[6898] := 16#935C;
   // GBK_TO_UNICODE[6899] := 16#63EC;
   // GBK_TO_UNICODE[6900] := 16#935D;
   // GBK_TO_UNICODE[6901] := 16#63EE;
   // GBK_TO_UNICODE[6902] := 16#935E;
   // GBK_TO_UNICODE[6903] := 16#63EF;
   // GBK_TO_UNICODE[6904] := 16#935F;
   // GBK_TO_UNICODE[6905] := 16#63F0;
   // GBK_TO_UNICODE[6906] := 16#9360;
   // GBK_TO_UNICODE[6907] := 16#63F1;
   // GBK_TO_UNICODE[6908] := 16#9361;
   // GBK_TO_UNICODE[6909] := 16#63F3;
   // GBK_TO_UNICODE[6910] := 16#9362;
   // GBK_TO_UNICODE[6911] := 16#63F5;
   // GBK_TO_UNICODE[6912] := 16#9363;
   // GBK_TO_UNICODE[6913] := 16#63F7;
   // GBK_TO_UNICODE[6914] := 16#9364;
   // GBK_TO_UNICODE[6915] := 16#63F9;
   // GBK_TO_UNICODE[6916] := 16#9365;
   // GBK_TO_UNICODE[6917] := 16#63FA;
   // GBK_TO_UNICODE[6918] := 16#9366;
   // GBK_TO_UNICODE[6919] := 16#63FB;
   // GBK_TO_UNICODE[6920] := 16#9367;
   // GBK_TO_UNICODE[6921] := 16#63FC;
   // GBK_TO_UNICODE[6922] := 16#9368;
   // GBK_TO_UNICODE[6923] := 16#63FE;
   // GBK_TO_UNICODE[6924] := 16#9369;
   // GBK_TO_UNICODE[6925] := 16#6403;
   // GBK_TO_UNICODE[6926] := 16#936A;
   // GBK_TO_UNICODE[6927] := 16#6404;
   // GBK_TO_UNICODE[6928] := 16#936B;
   // GBK_TO_UNICODE[6929] := 16#6406;
   // GBK_TO_UNICODE[6930] := 16#936C;
   // GBK_TO_UNICODE[6931] := 16#6407;
   // GBK_TO_UNICODE[6932] := 16#936D;
   // GBK_TO_UNICODE[6933] := 16#6408;
   // GBK_TO_UNICODE[6934] := 16#936E;
   // GBK_TO_UNICODE[6935] := 16#6409;
   // GBK_TO_UNICODE[6936] := 16#936F;
   // GBK_TO_UNICODE[6937] := 16#640A;
   // GBK_TO_UNICODE[6938] := 16#9370;
   // GBK_TO_UNICODE[6939] := 16#640D;
   // GBK_TO_UNICODE[6940] := 16#9371;
   // GBK_TO_UNICODE[6941] := 16#640E;
   // GBK_TO_UNICODE[6942] := 16#9372;
   // GBK_TO_UNICODE[6943] := 16#6411;
   // GBK_TO_UNICODE[6944] := 16#9373;
   // GBK_TO_UNICODE[6945] := 16#6412;
   // GBK_TO_UNICODE[6946] := 16#9374;
   // GBK_TO_UNICODE[6947] := 16#6415;
   // GBK_TO_UNICODE[6948] := 16#9375;
   // GBK_TO_UNICODE[6949] := 16#6416;
   // GBK_TO_UNICODE[6950] := 16#9376;
   // GBK_TO_UNICODE[6951] := 16#6417;
   // GBK_TO_UNICODE[6952] := 16#9377;
   // GBK_TO_UNICODE[6953] := 16#6418;
   // GBK_TO_UNICODE[6954] := 16#9378;
   // GBK_TO_UNICODE[6955] := 16#6419;
   // GBK_TO_UNICODE[6956] := 16#9379;
   // GBK_TO_UNICODE[6957] := 16#641A;
   // GBK_TO_UNICODE[6958] := 16#937A;
   // GBK_TO_UNICODE[6959] := 16#641D;
   // GBK_TO_UNICODE[6960] := 16#937B;
   // GBK_TO_UNICODE[6961] := 16#641F;
   // GBK_TO_UNICODE[6962] := 16#937C;
   // GBK_TO_UNICODE[6963] := 16#6422;
   // GBK_TO_UNICODE[6964] := 16#937D;
   // GBK_TO_UNICODE[6965] := 16#6423;
   // GBK_TO_UNICODE[6966] := 16#937E;
   // GBK_TO_UNICODE[6967] := 16#6424;
   // GBK_TO_UNICODE[6968] := 16#9380;
   // GBK_TO_UNICODE[6969] := 16#6425;
   // GBK_TO_UNICODE[6970] := 16#9381;
   // GBK_TO_UNICODE[6971] := 16#6427;
   // GBK_TO_UNICODE[6972] := 16#9382;
   // GBK_TO_UNICODE[6973] := 16#6428;
   // GBK_TO_UNICODE[6974] := 16#9383;
   // GBK_TO_UNICODE[6975] := 16#6429;
   // GBK_TO_UNICODE[6976] := 16#9384;
   // GBK_TO_UNICODE[6977] := 16#642B;
   // GBK_TO_UNICODE[6978] := 16#9385;
   // GBK_TO_UNICODE[6979] := 16#642E;
   // GBK_TO_UNICODE[6980] := 16#9386;
   // GBK_TO_UNICODE[6981] := 16#642F;
   // GBK_TO_UNICODE[6982] := 16#9387;
   // GBK_TO_UNICODE[6983] := 16#6430;
   // GBK_TO_UNICODE[6984] := 16#9388;
   // GBK_TO_UNICODE[6985] := 16#6431;
   // GBK_TO_UNICODE[6986] := 16#9389;
   // GBK_TO_UNICODE[6987] := 16#6432;
   // GBK_TO_UNICODE[6988] := 16#938A;
   // GBK_TO_UNICODE[6989] := 16#6433;
   // GBK_TO_UNICODE[6990] := 16#938B;
   // GBK_TO_UNICODE[6991] := 16#6435;
   // GBK_TO_UNICODE[6992] := 16#938C;
